LIN {X 0.182,Y -586.675,Z 1367.217,A 0.000,B 0.000,C 90.000,E1 75.102} C_DIS
LIN {X -0.131,Y -587.577,Z 1367.210,A 0.000,B 0.000,C 90.000,E1 73.795} C_DIS
LIN {X -0.025,Y -588.600,Z 1367.201,A 0.000,B 0.000,C 90.000,E1 72.181} C_DIS
LIN {X 0.175,Y -589.174,Z 1367.195,A 0.000,B 0.000,C 90.000,E1 71.094} C_DIS
LIN {X -0.190,Y -590.267,Z 1367.185,A 0.000,B 0.000,C 90.000,E1 69.263} C_DIS
LIN {X 0.230,Y -591.450,Z 1367.174,A 0.000,B 0.000,C 90.000,E1 67.358} C_DIS
LIN {X -0.084,Y -592.660,Z 1367.166,A 0.000,B 0.000,C 90.000,E1 65.793} C_DIS
LIN {X -0.029,Y -593.812,Z 1367.158,A 0.000,B 0.000,C 90.000,E1 64.460} C_DIS
LIN {X -0.046,Y -594.956,Z 1367.149,A 0.000,B 0.000,C 90.000,E1 62.871} C_DIS
LIN {X 0.337,Y -596.678,Z 1367.138,A 0.000,B 0.000,C 90.000,E1 60.717} C_DIS
LIN {X 0.286,Y -597.682,Z 1367.132,A 0.000,B 0.000,C 90.000,E1 59.665} C_DIS
LIN {X -0.217,Y -599.480,Z 1367.121,A 0.000,B 0.000,C 90.000,E1 57.867} C_DIS
LIN {X 0.070,Y -600.420,Z 1367.116,A 0.000,B 0.000,C 90.000,E1 56.786} C_DIS
LIN {X 0.111,Y -601.675,Z 1367.108,A 0.000,B 0.000,C 90.000,E1 55.468} C_DIS
LIN {X -0.317,Y -602.919,Z 1367.101,A 0.000,B 0.000,C 90.000,E1 54.196} C_DIS
LIN {X -0.207,Y -604.569,Z 1367.091,A 0.000,B 0.000,C 90.000,E1 52.351} C_DIS
LIN {X -0.112,Y -605.339,Z 1367.085,A 0.000,B 0.000,C 90.000,E1 51.295} C_DIS
LIN {X -0.057,Y -606.339,Z 1367.075,A 0.000,B 0.000,C 90.000,E1 49.461} C_DIS
LIN {X 0.070,Y -606.805,Z 1367.069,A 0.000,B 0.000,C 90.000,E1 48.405} C_DIS
LIN {X 0.003,Y -607.133,Z 1367.062,A 0.000,B 0.000,C 90.000,E1 47.106} C_DIS
LIN {X -0.086,Y -607.336,Z 1367.055,A 0.000,B 0.000,C 90.000,E1 45.810} C_DIS
LIN {X -0.164,Y -607.214,Z 1367.047,A 0.000,B 0.000,C 90.000,E1 44.514} C_DIS
LIN {X -0.060,Y -606.926,Z 1367.042,A 0.000,B 0.000,C 90.000,E1 43.461} C_DIS
LIN {X -0.317,Y -606.188,Z 1367.033,A 0.000,B 0.000,C 90.000,E1 41.919} C_DIS
LIN {X -0.191,Y -605.656,Z 1367.027,A 0.000,B 0.000,C 90.000,E1 40.862} C_DIS
LIN {X -0.274,Y -604.805,Z 1367.020,A 0.000,B 0.000,C 90.000,E1 39.564} C_DIS
LIN {X 0.036,Y -604.233,Z 1367.015,A 0.000,B 0.000,C 90.000,E1 38.749} C_DIS
LIN {X 0.006,Y -603.104,Z 1367.008,A 0.000,B 0.000,C 90.000,E1 37.443} C_DIS
LIN {X 0.185,Y -601.962,Z 1367.002,A 0.000,B 0.000,C 90.000,E1 36.377} C_DIS
LIN {X -0.151,Y -601.213,Z 1366.999,A 0.000,B 0.000,C 90.000,E1 35.884} C_DIS
LIN {X 0.000,Y -599.501,Z 1366.994,A 0.000,B 0.000,C 90.000,E1 34.818} C_DIS
LIN {X 0.014,Y -596.707,Z 1366.986,A 0.000,B 0.000,C 90.000,E1 33.499} C_DIS
LIN {X 0.259,Y -594.134,Z 1366.980,A 0.000,B 0.000,C 90.000,E1 32.418} C_DIS
LIN {X -0.241,Y -591.891,Z 1366.976,A 0.000,B 0.000,C 90.000,E1 31.671} C_DIS
LIN {X -0.146,Y -590.279,Z 1366.973,A 0.000,B 0.000,C 90.000,E1 31.131} C_DIS
LIN {X 0.001,Y -586.439,Z 1366.967,A 0.000,B 0.000,C 90.000,E1 30.050} C_DIS
LIN {X -0.076,Y -583.279,Z 1366.963,A 0.000,B 0.000,C 90.000,E1 29.255} C_DIS
LIN {X 0.110,Y -580.242,Z 1366.959,A 0.000,B 0.000,C 90.000,E1 28.565} C_DIS
LIN {X 0.037,Y -576.987,Z 1366.955,A 0.000,B 0.000,C 90.000,E1 27.897} C_DIS
LIN {X 0.097,Y -572.727,Z 1366.951,A 0.000,B 0.000,C 90.000,E1 27.078} C_DIS
LIN {X -0.054,Y -568.945,Z 1366.947,A 0.000,B 0.000,C 90.000,E1 26.411} C_DIS
LIN {X 0.018,Y -564.798,Z 1366.943,A 0.000,B 0.000,C 90.000,E1 25.720} C_DIS
LIN {X 0.152,Y -561.285,Z 1366.940,A 0.000,B 0.000,C 90.000,E1 25.155} C_DIS
LIN {X 0.054,Y -555.570,Z 1366.935,A 0.000,B 0.000,C 90.000,E1 24.335} C_DIS
LIN {X 0.134,Y -550.552,Z 1366.932,A 0.000,B 0.000,C 90.000,E1 23.643} C_DIS
LIN {X 0.165,Y -546.171,Z 1366.928,A 0.000,B 0.000,C 90.000,E1 23.078} C_DIS
LIN {X 0.114,Y -540.423,Z 1366.924,A 0.000,B 0.000,C 90.000,E1 22.386} C_DIS
LIN {X -0.268,Y -534.283,Z 1366.921,A 0.000,B 0.000,C 90.000,E1 21.716} C_DIS
LIN {X 0.001,Y -523.934,Z 1366.914,A 0.000,B 0.000,C 90.000,E1 20.556} C_DIS
LIN {X -0.191,Y -511.865,Z 1366.907,A 0.000,B 0.000,C 90.000,E1 19.322} C_DIS
LIN {X -0.080,Y -502.797,Z 1366.902,A 0.000,B 0.000,C 90.000,E1 18.362} C_DIS
LIN {X -0.238,Y -493.197,Z 1366.897,A 0.000,B 0.000,C 90.000,E1 17.402} C_DIS
LIN {X 0.136,Y -480.687,Z 1366.890,A 0.000,B 0.000,C 90.000,E1 16.134} C_DIS
LIN {X 0.231,Y -465.377,Z 1366.881,A 0.000,B 0.000,C 90.000,E1 14.592} C_DIS
LIN {X -0.148,Y -455.458,Z 1366.876,A 0.000,B 0.000,C 90.000,E1 13.647} C_DIS
LIN {X -0.104,Y -438.414,Z 1366.866,A 0.000,B 0.000,C 90.000,E1 11.883} C_DIS
LIN {X 0.074,Y -430.022,Z 1366.861,A 0.000,B 0.000,C 90.000,E1 10.950} C_DIS
LIN {X 0.023,Y -416.118,Z 1366.852,A 0.000,B 0.000,C 90.000,E1 9.378} C_DIS
LIN {X -0.121,Y -403.557,Z 1366.844,A 0.000,B 0.000,C 90.000,E1 7.936} C_DIS
LIN {X 0.155,Y -397.824,Z 1366.840,A 0.000,B 0.000,C 90.000,E1 7.239} C_DIS
LIN {X -0.185,Y -392.988,Z 1366.837,A 0.000,B 0.000,C 90.000,E1 6.606} C_DIS
LIN {X 0.034,Y -392.603,Z 1366.836,A 0.000,B 0.000,C 90.000,E1 6.486} C_DIS
LIN {X -0.004,Y -392.597,Z 1366.836,A 0.000,B 0.000,C 90.000,E1 6.486} C_DIS
LIN {X 0.166,Y -394.316,Z 1366.835,A 0.000,B 0.000,C 90.000,E1 6.201} C_DIS
LIN {X -0.174,Y -398.130,Z 1366.833,A 0.000,B 0.000,C 90.000,E1 5.910} C_DIS
LIN {X -0.140,Y -408.338,Z 1366.829,A 0.000,B 0.000,C 90.000,E1 5.163} C_DIS
LIN {X -0.103,Y -415.972,Z 1366.825,A 0.000,B 0.000,C 90.000,E1 4.531} C_DIS
LIN {X -0.114,Y -420.296,Z 1366.823,A 0.000,B 0.000,C 90.000,E1 4.131} C_DIS
LIN {X 0.071,Y -424.536,Z 1366.820,A 0.000,B 0.000,C 90.000,E1 3.669} C_DIS
LIN {X 0.122,Y -430.041,Z 1366.817,A 0.000,B 0.000,C 90.000,E1 3.037} C_DIS
LIN {X -0.080,Y -435.402,Z 1366.813,A 0.000,B 0.000,C 90.000,E1 2.407} C_DIS
LIN {X 0.212,Y -441.815,Z 1366.809,A 0.000,B 0.000,C 90.000,E1 1.547} C_DIS
LIN {X 0.086,Y -447.840,Z 1366.804,A 0.000,B 0.000,C 90.000,E1 0.745} C_DIS
LIN {X 0.000,Y -453.201,Z 1366.800,A 0.000,B 0.000,C 90.000,E1 360.000} C_DIS
LIN {X 0.073,Y -458.775,Z 1366.795,A 0.000,B 0.000,C 90.000,E1 359.141} C_DIS
LIN {X 0.003,Y -462.817,Z 1366.792,A 0.000,B 0.000,C 90.000,E1 358.511} C_DIS
LIN {X 0.204,Y -468.275,Z 1366.786,A 0.000,B 0.000,C 90.000,E1 357.535} C_DIS
LIN {X 0.203,Y -471.754,Z 1366.783,A 0.000,B 0.000,C 90.000,E1 356.906} C_DIS
LIN {X -0.091,Y -475.709,Z 1366.779,A 0.000,B 0.000,C 90.000,E1 356.159} C_DIS
LIN {X 0.125,Y -479.359,Z 1366.774,A 0.000,B 0.000,C 90.000,E1 355.355} C_DIS
LIN {X -0.101,Y -482.673,Z 1366.770,A 0.000,B 0.000,C 90.000,E1 354.609} C_DIS
LIN {X -0.109,Y -484.570,Z 1366.767,A 0.000,B 0.000,C 90.000,E1 354.147} C_DIS
LIN {X -0.093,Y -487.981,Z 1366.762,A 0.000,B 0.000,C 90.000,E1 353.223} C_DIS
LIN {X -0.039,Y -491.080,Z 1366.757,A 0.000,B 0.000,C 90.000,E1 352.299} C_DIS
LIN {X 0.226,Y -492.982,Z 1366.754,A 0.000,B 0.000,C 90.000,E1 351.659} C_DIS
LIN {X -0.054,Y -494.713,Z 1366.750,A 0.000,B 0.000,C 90.000,E1 351.084} C_DIS
LIN {X 0.154,Y -497.020,Z 1366.745,A 0.000,B 0.000,C 90.000,E1 350.151} C_DIS
LIN {X -0.096,Y -499.120,Z 1366.740,A 0.000,B 0.000,C 90.000,E1 349.275} C_DIS
LIN {X 0.096,Y -501.580,Z 1366.734,A 0.000,B 0.000,C 90.000,E1 348.049} C_DIS
LIN {X -0.042,Y -502.671,Z 1366.730,A 0.000,B 0.000,C 90.000,E1 347.465} C_DIS
LIN {X -0.183,Y -504.702,Z 1366.724,A 0.000,B 0.000,C 90.000,E1 346.284} C_DIS
LIN {X 0.187,Y -505.538,Z 1366.720,A 0.000,B 0.000,C 90.000,E1 345.644} C_DIS
LIN {X 0.127,Y -505.707,Z 1366.719,A 0.000,B 0.000,C 90.000,E1 345.353} C_DIS
LIN {X 0.198,Y -505.709,Z 1366.717,A 0.000,B 0.000,C 90.000,E1 345.046} C_DIS
LIN {X 0.139,Y -505.490,Z 1366.715,A 0.000,B 0.000,C 90.000,E1 344.755} C_DIS
LIN {X 0.078,Y -504.841,Z 1366.714,A 0.000,B 0.000,C 90.000,E1 344.464} C_DIS
LIN {X -0.128,Y -504.230,Z 1366.713,A 0.000,B 0.000,C 90.000,E1 344.338} C_DIS
LIN {X 0.152,Y -503.084,Z 1366.712,A 0.000,B 0.000,C 90.000,E1 344.157} C_DIS
LIN {X 0.156,Y -499.851,Z 1366.711,A 0.000,B 0.000,C 90.000,E1 344.031} C_DIS
LIN {X -0.040,Y -466.644,Z 1366.705,A 0.000,B 0.000,C 90.000,E1 342.906} C_DIS
LIN {X 0.169,Y -435.494,Z 1366.698,A 0.000,B 0.000,C 90.000,E1 341.638} C_DIS
LIN {X -0.147,Y -408.031,Z 1366.691,A 0.000,B 0.000,C 90.000,E1 340.423} C_DIS
LIN {X -0.120,Y -382.486,Z 1366.684,A 0.000,B 0.000,C 90.000,E1 339.082} C_DIS
LIN {X 0.064,Y -362.176,Z 1366.677,A 0.000,B 0.000,C 90.000,E1 337.847} C_DIS
LIN {X 0.043,Y -362.174,Z 1366.677,A 0.000,B 0.000,C 90.000,E1 337.847} C_DIS
LIN {X 0.164,Y -366.198,Z 1366.641,A 0.000,B 0.000,C 90.000,E1 331.385} C_DIS
LIN {X -0.133,Y -371.227,Z 1366.604,A 0.000,B 0.000,C 90.000,E1 324.769} C_DIS
LIN {X -0.146,Y -371.660,Z 1366.602,A 0.000,B 0.000,C 90.000,E1 324.402} C_DIS
LIN {X -0.090,Y -376.765,Z 1366.570,A 0.000,B 0.000,C 90.000,E1 318.528} C_DIS
LIN {X 0.200,Y -378.156,Z 1366.563,A 0.000,B 0.000,C 90.000,E1 317.391} C_DIS
LIN {X -0.061,Y -384.283,Z 1366.529,A 0.000,B 0.000,C 90.000,E1 311.272} C_DIS
LIN {X -0.019,Y -384.786,Z 1366.527,A 0.000,B 0.000,C 90.000,E1 310.906} C_DIS
LIN {X -0.029,Y -390.954,Z 1366.493,A 0.000,B 0.000,C 90.000,E1 304.818} C_DIS
LIN {X 0.038,Y -391.366,Z 1366.491,A 0.000,B 0.000,C 90.000,E1 304.452} C_DIS
LIN {X -0.232,Y -396.686,Z 1366.460,A 0.000,B 0.000,C 90.000,E1 298.821} C_DIS
LIN {X -0.014,Y -397.074,Z 1366.458,A 0.000,B 0.000,C 90.000,E1 298.437} C_DIS
LIN {X -0.058,Y -401.487,Z 1366.427,A 0.000,B 0.000,C 90.000,E1 292.823} C_DIS
LIN {X 0.108,Y -401.768,Z 1366.423,A 0.000,B 0.000,C 90.000,E1 292.099} C_DIS
LIN {X 0.068,Y -404.565,Z 1366.396,A 0.000,B 0.000,C 90.000,E1 287.221} C_DIS
LIN {X 0.170,Y -404.760,Z 1366.394,A 0.000,B 0.000,C 90.000,E1 286.858} C_DIS
LIN {X 0.077,Y -406.039,Z 1366.365,A 0.000,B 0.000,C 90.000,E1 281.658} C_DIS
LIN {X 0.166,Y -406.138,Z 1366.363,A 0.000,B 0.000,C 90.000,E1 281.299} C_DIS
LIN {X -0.207,Y -405.655,Z 1366.334,A 0.000,B 0.000,C 90.000,E1 276.144} C_DIS
LIN {X 0.201,Y -405.601,Z 1366.332,A 0.000,B 0.000,C 90.000,E1 275.739} C_DIS
LIN {X -0.129,Y -403.549,Z 1366.305,A 0.000,B 0.000,C 90.000,E1 270.917} C_DIS
LIN {X -0.194,Y -403.040,Z 1366.301,A 0.000,B 0.000,C 90.000,E1 270.229} C_DIS
LIN {X 0.031,Y -399.011,Z 1366.272,A 0.000,B 0.000,C 90.000,E1 264.951} C_DIS
LIN {X -0.143,Y -397.175,Z 1366.264,A 0.000,B 0.000,C 90.000,E1 263.571} C_DIS
LIN {X -0.194,Y -392.923,Z 1366.241,A 0.000,B 0.000,C 90.000,E1 259.342} C_DIS
LIN {X 0.182,Y -391.869,Z 1366.237,A 0.000,B 0.000,C 90.000,E1 258.578} C_DIS
LIN {X -0.062,Y -385.732,Z 1366.211,A 0.000,B 0.000,C 90.000,E1 253.976} C_DIS
LIN {X -0.127,Y -384.968,Z 1366.207,A 0.000,B 0.000,C 90.000,E1 253.268} C_DIS
LIN {X 0.100,Y -378.113,Z 1366.183,A 0.000,B 0.000,C 90.000,E1 248.901} C_DIS
LIN {X -0.164,Y -376.355,Z 1366.175,A 0.000,B 0.000,C 90.000,E1 247.486} C_DIS
LIN {X -0.038,Y -375.852,Z 1366.173,A 0.000,B 0.000,C 90.000,E1 247.102} C_DIS
LIN {X -0.088,Y -369.083,Z 1366.150,A 0.000,B 0.000,C 90.000,E1 243.076} C_DIS
LIN {X -0.009,Y -366.236,Z 1366.138,A 0.000,B 0.000,C 90.000,E1 240.845} C_DIS
LIN {X -0.047,Y -358.830,Z 1366.113,A 0.000,B 0.000,C 90.000,E1 236.373} C_DIS
LIN {X -0.059,Y -356.022,Z 1366.101,A 0.000,B 0.000,C 90.000,E1 234.116} C_DIS
LIN {X -0.062,Y -348.459,Z 1366.073,A 0.000,B 0.000,C 90.000,E1 229.175} C_DIS
LIN {X -0.001,Y -345.873,Z 1366.060,A 0.000,B 0.000,C 90.000,E1 226.863} C_DIS
LIN {X -0.033,Y -339.106,Z 1366.032,A 0.000,B 0.000,C 90.000,E1 221.838} C_DIS
LIN {X 0.051,Y -336.944,Z 1366.019,A 0.000,B 0.000,C 90.000,E1 219.483} C_DIS
LIN {X 0.031,Y -331.620,Z 1365.993,A 0.000,B 0.000,C 90.000,E1 214.771} C_DIS
LIN {X 0.101,Y -329.361,Z 1365.976,A 0.000,B 0.000,C 90.000,E1 211.592} C_DIS
LIN {X 0.113,Y -328.630,Z 1365.971,A 0.000,B 0.000,C 90.000,E1 210.797} C_DIS
LIN {X -0.181,Y -324.550,Z 1365.940,A 0.000,B 0.000,C 90.000,E1 205.283} C_DIS
LIN {X -0.199,Y -324.574,Z 1365.940,A 0.000,B 0.000,C 90.000,E1 205.283} C_DIS
LIN {X -0.065,Y -343.510,Z 1365.932,A 0.000,B 0.000,C 90.000,E1 203.823} C_DIS
LIN {X 0.111,Y -364.170,Z 1365.925,A 0.000,B 0.000,C 90.000,E1 202.408} C_DIS
LIN {X -0.078,Y -386.764,Z 1365.917,A 0.000,B 0.000,C 90.000,E1 201.099} C_DIS
LIN {X 0.144,Y -413.035,Z 1365.910,A 0.000,B 0.000,C 90.000,E1 199.704} C_DIS
LIN {X 0.218,Y -441.275,Z 1365.902,A 0.000,B 0.000,C 90.000,E1 198.417} C_DIS
LIN {X -0.100,Y -446.323,Z 1365.901,A 0.000,B 0.000,C 90.000,E1 198.236} C_DIS
LIN {X 0.088,Y -447.679,Z 1365.900,A 0.000,B 0.000,C 90.000,E1 198.055} C_DIS
LIN {X 0.266,Y -448.506,Z 1365.900,A 0.000,B 0.000,C 90.000,E1 197.873} C_DIS
LIN {X -0.122,Y -449.127,Z 1365.899,A 0.000,B 0.000,C 90.000,E1 197.764} C_DIS
LIN {X 0.177,Y -450.069,Z 1365.897,A 0.000,B 0.000,C 90.000,E1 197.402} C_DIS
LIN {X 0.048,Y -450.694,Z 1365.895,A 0.000,B 0.000,C 90.000,E1 197.094} C_DIS
LIN {X -0.210,Y -451.133,Z 1365.893,A 0.000,B 0.000,C 90.000,E1 196.804} C_DIS
LIN {X 0.155,Y -451.880,Z 1365.888,A 0.000,B 0.000,C 90.000,E1 195.788} C_DIS
LIN {X 0.045,Y -453.011,Z 1365.879,A 0.000,B 0.000,C 90.000,E1 194.189} C_DIS
LIN {X 0.188,Y -453.802,Z 1365.872,A 0.000,B 0.000,C 90.000,E1 192.883} C_DIS
LIN {X -0.002,Y -454.650,Z 1365.863,A 0.000,B 0.000,C 90.000,E1 191.299} C_DIS
LIN {X -0.036,Y -455.227,Z 1365.856,A 0.000,B 0.000,C 90.000,E1 190.018} C_DIS
LIN {X -0.134,Y -455.673,Z 1365.849,A 0.000,B 0.000,C 90.000,E1 188.746} C_DIS
LIN {X 0.075,Y -455.919,Z 1365.843,A 0.000,B 0.000,C 90.000,E1 187.757} C_DIS
LIN {X -0.081,Y -456.266,Z 1365.833,A 0.000,B 0.000,C 90.000,E1 185.853} C_DIS
LIN {X 0.028,Y -456.324,Z 1365.827,A 0.000,B 0.000,C 90.000,E1 184.878} C_DIS
LIN {X -0.101,Y -456.190,Z 1365.820,A 0.000,B 0.000,C 90.000,E1 183.612} C_DIS
LIN {X 0.011,Y -455.960,Z 1365.815,A 0.000,B 0.000,C 90.000,E1 182.636} C_DIS
LIN {X -0.080,Y -455.745,Z 1365.811,A 0.000,B 0.000,C 90.000,E1 182.007} C_DIS
LIN {X 0.023,Y -455.119,Z 1365.806,A 0.000,B 0.000,C 90.000,E1 181.031} C_DIS
LIN {X -0.072,Y -454.546,Z 1365.802,A 0.000,B 0.000,C 90.000,E1 180.401} C_DIS
LIN {X -0.169,Y -453.770,Z 1365.799,A 0.000,B 0.000,C 90.000,E1 179.771} C_DIS
LIN {X 0.067,Y -451.689,Z 1365.792,A 0.000,B 0.000,C 90.000,E1 178.453} C_DIS
LIN {X -0.039,Y -450.487,Z 1365.788,A 0.000,B 0.000,C 90.000,E1 177.822} C_DIS
LIN {X 0.123,Y -449.773,Z 1365.786,A 0.000,B 0.000,C 90.000,E1 177.478} C_DIS
LIN {X -0.169,Y -448.926,Z 1365.784,A 0.000,B 0.000,C 90.000,E1 177.192} C_DIS
LIN {X -0.144,Y -445.871,Z 1365.779,A 0.000,B 0.000,C 90.000,E1 176.216} C_DIS
LIN {X 0.158,Y -443.707,Z 1365.775,A 0.000,B 0.000,C 90.000,E1 175.527} C_DIS
LIN {X 0.000,Y -440.751,Z 1365.772,A 0.000,B 0.000,C 90.000,E1 174.894} C_DIS
LIN {X 0.204,Y -438.571,Z 1365.769,A 0.000,B 0.000,C 90.000,E1 174.375} C_DIS
LIN {X 0.049,Y -434.159,Z 1365.764,A 0.000,B 0.000,C 90.000,E1 173.571} C_DIS
LIN {X -0.218,Y -431.237,Z 1365.762,A 0.000,B 0.000,C 90.000,E1 173.109} C_DIS
LIN {X 0.032,Y -425.872,Z 1365.757,A 0.000,B 0.000,C 90.000,E1 172.243} C_DIS
LIN {X -0.194,Y -420.132,Z 1365.752,A 0.000,B 0.000,C 90.000,E1 171.432} C_DIS
LIN {X 0.101,Y -406.286,Z 1365.741,A 0.000,B 0.000,C 90.000,E1 169.342} C_DIS
LIN {X 0.216,Y -393.490,Z 1365.729,A 0.000,B 0.000,C 90.000,E1 167.229} C_DIS
LIN {X 0.198,Y -390.708,Z 1365.726,A 0.000,B 0.000,C 90.000,E1 166.700} C_DIS
LIN {X -0.069,Y -387.799,Z 1365.722,A 0.000,B 0.000,C 90.000,E1 165.936} C_DIS
LIN {X -0.087,Y -387.536,Z 1365.719,A 0.000,B 0.000,C 90.000,E1 165.408} C_DIS
LIN {X -0.125,Y -387.556,Z 1365.719,A 0.000,B 0.000,C 90.000,E1 165.408} C_DIS
LIN {X -0.135,Y -388.274,Z 1365.718,A 0.000,B 0.000,C 90.000,E1 165.227} C_DIS
LIN {X -0.128,Y -392.971,Z 1365.714,A 0.000,B 0.000,C 90.000,E1 164.574} C_DIS
LIN {X -0.108,Y -399.230,Z 1365.710,A 0.000,B 0.000,C 90.000,E1 163.866} C_DIS
LIN {X -0.180,Y -408.697,Z 1365.705,A 0.000,B 0.000,C 90.000,E1 162.960} C_DIS
LIN {X 0.013,Y -425.885,Z 1365.697,A 0.000,B 0.000,C 90.000,E1 161.456} C_DIS
LIN {X 0.257,Y -449.800,Z 1365.687,A 0.000,B 0.000,C 90.000,E1 159.571} C_DIS
LIN {X -0.100,Y -459.141,Z 1365.683,A 0.000,B 0.000,C 90.000,E1 158.901} C_DIS
LIN {X -0.021,Y -466.703,Z 1365.679,A 0.000,B 0.000,C 90.000,E1 158.284} C_DIS
LIN {X -0.108,Y -472.655,Z 1365.677,A 0.000,B 0.000,C 90.000,E1 157.794} C_DIS
LIN {X -0.283,Y -481.389,Z 1365.672,A 0.000,B 0.000,C 90.000,E1 157.050} C_DIS
LIN {X -0.124,Y -489.927,Z 1365.668,A 0.000,B 0.000,C 90.000,E1 156.230} C_DIS
LIN {X 0.098,Y -495.512,Z 1365.665,A 0.000,B 0.000,C 90.000,E1 155.665} C_DIS
LIN {X 0.218,Y -500.943,Z 1365.662,A 0.000,B 0.000,C 90.000,E1 155.101} C_DIS
LIN {X -0.117,Y -504.951,Z 1365.660,A 0.000,B 0.000,C 90.000,E1 154.717} C_DIS
LIN {X -0.091,Y -512.632,Z 1365.655,A 0.000,B 0.000,C 90.000,E1 153.845} C_DIS
LIN {X -0.256,Y -518.709,Z 1365.651,A 0.000,B 0.000,C 90.000,E1 153.127} C_DIS
LIN {X 0.082,Y -524.193,Z 1365.646,A 0.000,B 0.000,C 90.000,E1 152.359} C_DIS
LIN {X -0.238,Y -526.299,Z 1365.645,A 0.000,B 0.000,C 90.000,E1 152.103} C_DIS
LIN {X -0.145,Y -530.043,Z 1365.642,A 0.000,B 0.000,C 90.000,E1 151.513} C_DIS
LIN {X -0.170,Y -533.906,Z 1365.638,A 0.000,B 0.000,C 90.000,E1 150.795} C_DIS
LIN {X -0.019,Y -536.557,Z 1365.635,A 0.000,B 0.000,C 90.000,E1 150.205} C_DIS
LIN {X 0.144,Y -539.972,Z 1365.630,A 0.000,B 0.000,C 90.000,E1 149.331} C_DIS
LIN {X -0.127,Y -541.955,Z 1365.627,A 0.000,B 0.000,C 90.000,E1 148.791} C_DIS
LIN {X 0.079,Y -543.704,Z 1365.623,A 0.000,B 0.000,C 90.000,E1 148.201} C_DIS
LIN {X -0.140,Y -545.900,Z 1365.619,A 0.000,B 0.000,C 90.000,E1 147.375} C_DIS
LIN {X 0.089,Y -547.150,Z 1365.616,A 0.000,B 0.000,C 90.000,E1 146.786} C_DIS
LIN {X -0.049,Y -549.147,Z 1365.609,A 0.000,B 0.000,C 90.000,E1 145.674} C_DIS
LIN {X 0.106,Y -550.435,Z 1365.605,A 0.000,B 0.000,C 90.000,E1 144.815} C_DIS
LIN {X 0.017,Y -551.761,Z 1365.598,A 0.000,B 0.000,C 90.000,E1 143.703} C_DIS
LIN {X 0.269,Y -552.794,Z 1365.592,A 0.000,B 0.000,C 90.000,E1 142.557} C_DIS
LIN {X 0.099,Y -553.616,Z 1365.586,A 0.000,B 0.000,C 90.000,E1 141.457} C_DIS
LIN {X 0.076,Y -554.674,Z 1365.577,A 0.000,B 0.000,C 90.000,E1 139.784} C_DIS
LIN {X -0.068,Y -555.526,Z 1365.569,A 0.000,B 0.000,C 90.000,E1 138.405} C_DIS
LIN {X -0.162,Y -556.345,Z 1365.560,A 0.000,B 0.000,C 90.000,E1 136.743} C_DIS
LIN {X 0.107,Y -556.913,Z 1365.552,A 0.000,B 0.000,C 90.000,E1 135.324} C_DIS
LIN {X 0.093,Y -557.710,Z 1365.541,A 0.000,B 0.000,C 90.000,E1 133.380} C_DIS
LIN {X 0.113,Y -558.710,Z 1365.530,A 0.000,B 0.000,C 90.000,E1 131.434} C_DIS
LIN {X -0.271,Y -559.658,Z 1365.526,A 0.000,B 0.000,C 90.000,E1 130.620} C_DIS
LIN {X -0.312,Y -559.675,Z 1365.526,A 0.000,B 0.000,C 90.000,E1 130.620} C_DIS
LIN {X 0.204,Y -560.719,Z 1365.525,A 0.000,B 0.000,C 90.000,E1 130.458} C_DIS
LIN {X 0.111,Y -561.623,Z 1365.524,A 0.000,B 0.000,C 90.000,E1 130.334} C_DIS
LIN {X 0.127,Y -562.227,Z 1365.523,A 0.000,B 0.000,C 90.000,E1 130.172} C_DIS
LIN {X 0.084,Y -562.282,Z 1365.523,A 0.000,B 0.000,C 90.000,E1 130.172} C_DIS
LIN {X -0.227,Y -564.588,Z 1365.523,A 0.000,B 0.000,C 90.000,E1 130.092} C_DIS
LIN {X -0.283,Y -566.188,Z 1365.522,A 0.000,B 0.000,C 90.000,E1 130.011} C_DIS
LIN {X 0.133,Y -574.296,Z 1365.521,A 0.000,B 0.000,C 90.000,E1 129.725} C_DIS
LIN {X 0.261,Y -579.457,Z 1365.520,A 0.000,B 0.000,C 90.000,E1 129.564} C_DIS
LIN {X 0.015,Y -581.996,Z 1365.519,A 0.000,B 0.000,C 90.000,E1 129.483} C_DIS
LIN {X -0.148,Y -585.029,Z 1365.519,A 0.000,B 0.000,C 90.000,E1 129.358} C_DIS
LIN {X 0.191,Y -590.891,Z 1365.517,A 0.000,B 0.000,C 90.000,E1 128.991} C_DIS
LIN {X -0.248,Y -595.306,Z 1365.515,A 0.000,B 0.000,C 90.000,E1 128.749} C_DIS
LIN {X 0.028,Y -600.950,Z 1365.513,A 0.000,B 0.000,C 90.000,E1 128.302} C_DIS
LIN {X 0.020,Y -606.411,Z 1365.510,A 0.000,B 0.000,C 90.000,E1 127.855} C_DIS
LIN {X -0.070,Y -612.969,Z 1365.507,A 0.000,B 0.000,C 90.000,E1 127.282} C_DIS
LIN {X -0.062,Y -616.756,Z 1365.505,A 0.000,B 0.000,C 90.000,E1 126.916} C_DIS
LIN {X 0.200,Y -625.260,Z 1365.500,A 0.000,B 0.000,C 90.000,E1 126.011} C_DIS
LIN {X -0.098,Y -628.604,Z 1365.498,A 0.000,B 0.000,C 90.000,E1 125.678} C_DIS
LIN {X 0.102,Y -635.118,Z 1365.494,A 0.000,B 0.000,C 90.000,E1 124.898} C_DIS
LIN {X -0.011,Y -640.076,Z 1365.490,A 0.000,B 0.000,C 90.000,E1 124.278} C_DIS
LIN {X 0.098,Y -643.801,Z 1365.488,A 0.000,B 0.000,C 90.000,E1 123.785} C_DIS
LIN {X 0.058,Y -648.265,Z 1365.484,A 0.000,B 0.000,C 90.000,E1 123.166} C_DIS
LIN {X 0.051,Y -652.359,Z 1365.481,A 0.000,B 0.000,C 90.000,E1 122.546} C_DIS
LIN {X -0.369,Y -654.670,Z 1365.479,A 0.000,B 0.000,C 90.000,E1 122.212} C_DIS
LIN {X -0.133,Y -658.591,Z 1365.475,A 0.000,B 0.000,C 90.000,E1 121.465} C_DIS
LIN {X 0.040,Y -660.427,Z 1365.473,A 0.000,B 0.000,C 90.000,E1 121.082} C_DIS
LIN {X 0.188,Y -663.616,Z 1365.469,A 0.000,B 0.000,C 90.000,E1 120.335} C_DIS
LIN {X 0.029,Y -666.155,Z 1365.465,A 0.000,B 0.000,C 90.000,E1 119.617} C_DIS
LIN {X 0.221,Y -668.142,Z 1365.461,A 0.000,B 0.000,C 90.000,E1 118.871} C_DIS
LIN {X 0.375,Y -668.696,Z 1365.459,A 0.000,B 0.000,C 90.000,E1 118.615} C_DIS
LIN {X 0.263,Y -669.704,Z 1365.455,A 0.000,B 0.000,C 90.000,E1 117.897} C_DIS
LIN {X -0.147,Y -669.966,Z 1365.451,A 0.000,B 0.000,C 90.000,E1 117.206} C_DIS
LIN {X -0.247,Y -669.843,Z 1365.447,A 0.000,B 0.000,C 90.000,E1 116.488} C_DIS
LIN {X 0.248,Y -669.374,Z 1365.443,A 0.000,B 0.000,C 90.000,E1 115.720} C_DIS
LIN {X -0.154,Y -668.585,Z 1365.439,A 0.000,B 0.000,C 90.000,E1 115.027} C_DIS
LIN {X 0.006,Y -668.253,Z 1365.438,A 0.000,B 0.000,C 90.000,E1 114.771} C_DIS
LIN {X 0.047,Y -666.989,Z 1365.435,A 0.000,B 0.000,C 90.000,E1 114.283} C_DIS
LIN {X 0.203,Y -666.014,Z 1365.434,A 0.000,B 0.000,C 90.000,E1 114.027} C_DIS
LIN {X -0.109,Y -663.067,Z 1365.431,A 0.000,B 0.000,C 90.000,E1 113.567} C_DIS
LIN {X -0.040,Y -662.029,Z 1365.430,A 0.000,B 0.000,C 90.000,E1 113.439} C_DIS
LIN {X -0.147,Y -656.469,Z 1365.428,A 0.000,B 0.000,C 90.000,E1 113.003} C_DIS
LIN {X -0.180,Y -654.733,Z 1365.427,A 0.000,B 0.000,C 90.000,E1 112.898} C_DIS
LIN {X -0.185,Y -648.596,Z 1365.426,A 0.000,B 0.000,C 90.000,E1 112.642} C_DIS
LIN {X -0.187,Y -644.606,Z 1365.425,A 0.000,B 0.000,C 90.000,E1 112.514} C_DIS
LIN {X -0.066,Y -634.954,Z 1365.424,A 0.000,B 0.000,C 90.000,E1 112.259} C_DIS
LIN {X 0.181,Y -629.604,Z 1365.423,A 0.000,B 0.000,C 90.000,E1 112.099} C_DIS
LIN {X 0.126,Y -629.435,Z 1365.423,A 0.000,B 0.000,C 90.000,E1 112.099} C_DIS
LIN {X -0.146,Y -630.466,Z 1365.422,A 0.000,B 0.000,C 90.000,E1 111.972} C_DIS
LIN {X -0.274,Y -639.281,Z 1365.416,A 0.000,B 0.000,C 90.000,E1 110.972} C_DIS
LIN {X -0.179,Y -643.249,Z 1365.414,A 0.000,B 0.000,C 90.000,E1 110.482} C_DIS
LIN {X 0.343,Y -647.430,Z 1365.410,A 0.000,B 0.000,C 90.000,E1 109.812} C_DIS
LIN {X 0.224,Y -649.628,Z 1365.408,A 0.000,B 0.000,C 90.000,E1 109.450} C_DIS
LIN {X -0.022,Y -653.008,Z 1365.405,A 0.000,B 0.000,C 90.000,E1 108.852} C_DIS
LIN {X -0.117,Y -657.558,Z 1365.399,A 0.000,B 0.000,C 90.000,E1 107.873} C_DIS
LIN {X 0.372,Y -660.755,Z 1365.395,A 0.000,B 0.000,C 90.000,E1 107.094} C_DIS
LIN {X 0.072,Y -663.615,Z 1365.391,A 0.000,B 0.000,C 90.000,E1 106.386} C_DIS
LIN {X -0.013,Y -666.033,Z 1365.387,A 0.000,B 0.000,C 90.000,E1 105.662} C_DIS
LIN {X -0.258,Y -667.873,Z 1365.383,A 0.000,B 0.000,C 90.000,E1 104.954} C_DIS
LIN {X 0.238,Y -668.850,Z 1365.380,A 0.000,B 0.000,C 90.000,E1 104.426} C_DIS
LIN {X 0.027,Y -669.855,Z 1365.376,A 0.000,B 0.000,C 90.000,E1 103.716} C_DIS
LIN {X -0.110,Y -670.297,Z 1365.374,A 0.000,B 0.000,C 90.000,E1 103.244} C_DIS
LIN {X -0.311,Y -670.497,Z 1365.370,A 0.000,B 0.000,C 90.000,E1 102.535} C_DIS
LIN {X 0.141,Y -670.333,Z 1365.365,A 0.000,B 0.000,C 90.000,E1 101.771} C_DIS
LIN {X 0.072,Y -670.208,Z 1365.364,A 0.000,B 0.000,C 90.000,E1 101.535} C_DIS
LIN {X -0.272,Y -669.384,Z 1365.360,A 0.000,B 0.000,C 90.000,E1 100.838} C_DIS
LIN {X 0.237,Y -668.657,Z 1365.357,A 0.000,B 0.000,C 90.000,E1 100.310} C_DIS
LIN {X -0.036,Y -667.668,Z 1365.355,A 0.000,B 0.000,C 90.000,E1 99.849} C_DIS
LIN {X -0.201,Y -666.410,Z 1365.352,A 0.000,B 0.000,C 90.000,E1 99.378} C_DIS
LIN {X 0.172,Y -664.934,Z 1365.349,A 0.000,B 0.000,C 90.000,E1 98.859} C_DIS
LIN {X -0.217,Y -662.224,Z 1365.345,A 0.000,B 0.000,C 90.000,E1 98.163} C_DIS
LIN {X 0.135,Y -660.250,Z 1365.343,A 0.000,B 0.000,C 90.000,E1 97.644} C_DIS
LIN {X -0.302,Y -656.924,Z 1365.339,A 0.000,B 0.000,C 90.000,E1 96.947} C_DIS
LIN {X 0.043,Y -655.113,Z 1365.336,A 0.000,B 0.000,C 90.000,E1 96.549} C_DIS
LIN {X -0.303,Y -652.457,Z 1365.334,A 0.000,B 0.000,C 90.000,E1 96.087} C_DIS
LIN {X -0.178,Y -647.963,Z 1365.330,A 0.000,B 0.000,C 90.000,E1 95.334} C_DIS
LIN {X -0.164,Y -643.191,Z 1365.325,A 0.000,B 0.000,C 90.000,E1 94.588} C_DIS
LIN {X -0.074,Y -638.959,Z 1365.322,A 0.000,B 0.000,C 90.000,E1 93.955} C_DIS
LIN {X 0.065,Y -635.128,Z 1365.319,A 0.000,B 0.000,C 90.000,E1 93.440} C_DIS
LIN {X 0.082,Y -629.543,Z 1365.316,A 0.000,B 0.000,C 90.000,E1 92.808} C_DIS
LIN {X 0.146,Y -623.401,Z 1365.312,A 0.000,B 0.000,C 90.000,E1 92.178} C_DIS
LIN {X 0.218,Y -615.720,Z 1365.308,A 0.000,B 0.000,C 90.000,E1 91.432} C_DIS
LIN {X -0.008,Y -611.713,Z 1365.306,A 0.000,B 0.000,C 90.000,E1 91.088} C_DIS
LIN {X -0.109,Y -607.317,Z 1365.304,A 0.000,B 0.000,C 90.000,E1 90.745} C_DIS
LIN {X 0.085,Y -602.939,Z 1365.302,A 0.000,B 0.000,C 90.000,E1 90.401} C_DIS
LIN {X 0.229,Y -596.196,Z 1365.300,A 0.000,B 0.000,C 90.000,E1 90.000} C_DIS
LIN {X -0.222,Y -589.332,Z 1365.298,A 0.000,B 0.000,C 90.000,E1 89.714} C_DIS
LIN {X -0.119,Y -584.030,Z 1365.297,A 0.000,B 0.000,C 90.000,E1 89.484} C_DIS
LIN {X 0.001,Y -578.143,Z 1365.296,A 0.000,B 0.000,C 90.000,E1 89.198} C_DIS
LIN {X -0.114,Y -574.268,Z 1365.294,A 0.000,B 0.000,C 90.000,E1 88.912} C_DIS
LIN {X -0.151,Y -574.243,Z 1365.294,A 0.000,B 0.000,C 90.000,E1 88.912} C_DIS
LIN {X -0.170,Y -573.640,Z 1365.293,A 0.000,B 0.000,C 90.000,E1 88.740} C_DIS
LIN {X -0.152,Y -573.457,Z 1365.292,A 0.000,B 0.000,C 90.000,E1 88.568} C_DIS
LIN {X -0.271,Y -573.745,Z 1365.288,A 0.000,B 0.000,C 90.000,E1 87.822} C_DIS
LIN {X -0.071,Y -575.894,Z 1365.274,A 0.000,B 0.000,C 90.000,E1 85.355} C_DIS
LIN {X -0.209,Y -577.628,Z 1365.265,A 0.000,B 0.000,C 90.000,E1 83.742} C_DIS
LIN {X -0.097,Y -579.909,Z 1365.255,A 0.000,B 0.000,C 90.000,E1 81.837} C_DIS
LIN {X 0.016,Y -581.829,Z 1365.246,A 0.000,B 0.000,C 90.000,E1 80.208} C_DIS
LIN {X 0.273,Y -583.045,Z 1365.240,A 0.000,B 0.000,C 90.000,E1 79.106} C_DIS
LIN {X 0.083,Y -584.087,Z 1365.234,A 0.000,B 0.000,C 90.000,E1 78.049} C_DIS
LIN {X 0.154,Y -585.375,Z 1365.226,A 0.000,B 0.000,C 90.000,E1 76.700} C_DIS
LIN {X -0.007,Y -586.218,Z 1365.220,A 0.000,B 0.000,C 90.000,E1 75.644} C_DIS
LIN {X 0.228,Y -587.178,Z 1365.213,A 0.000,B 0.000,C 90.000,E1 74.283} C_DIS
LIN {X 0.173,Y -588.365,Z 1365.203,A 0.000,B 0.000,C 90.000,E1 72.417} C_DIS
LIN {X 0.185,Y -588.987,Z 1365.197,A 0.000,B 0.000,C 90.000,E1 71.348} C_DIS
LIN {X -0.196,Y -590.030,Z 1365.186,A 0.000,B 0.000,C 90.000,E1 69.518} C_DIS
LIN {X -0.224,Y -591.014,Z 1365.177,A 0.000,B 0.000,C 90.000,E1 67.922} C_DIS
LIN {X -0.113,Y -592.384,Z 1365.167,A 0.000,B 0.000,C 90.000,E1 66.049} C_DIS
LIN {X -0.161,Y -593.741,Z 1365.158,A 0.000,B 0.000,C 90.000,E1 64.460} C_DIS
LIN {X -0.180,Y -594.893,Z 1365.149,A 0.000,B 0.000,C 90.000,E1 62.871} C_DIS
LIN {X -0.001,Y -596.374,Z 1365.139,A 0.000,B 0.000,C 90.000,E1 61.001} C_DIS
LIN {X 0.151,Y -597.626,Z 1365.132,A 0.000,B 0.000,C 90.000,E1 59.665} C_DIS
LIN {X -0.267,Y -599.147,Z 1365.123,A 0.000,B 0.000,C 90.000,E1 58.122} C_DIS
LIN {X 0.022,Y -600.163,Z 1365.117,A 0.000,B 0.000,C 90.000,E1 57.041} C_DIS
LIN {X 0.065,Y -601.391,Z 1365.110,A 0.000,B 0.000,C 90.000,E1 55.722} C_DIS
LIN {X 0.031,Y -602.853,Z 1365.101,A 0.000,B 0.000,C 90.000,E1 54.149} C_DIS
LIN {X 0.238,Y -604.303,Z 1365.092,A 0.000,B 0.000,C 90.000,E1 52.557} C_DIS
LIN {X -0.045,Y -605.097,Z 1365.086,A 0.000,B 0.000,C 90.000,E1 51.537} C_DIS
LIN {X -0.060,Y -605.855,Z 1365.079,A 0.000,B 0.000,C 90.000,E1 50.231} C_DIS
LIN {X 0.058,Y -606.439,Z 1365.073,A 0.000,B 0.000,C 90.000,E1 49.175} C_DIS
LIN {X -0.271,Y -606.824,Z 1365.068,A 0.000,B 0.000,C 90.000,E1 48.162} C_DIS
LIN {X 0.081,Y -607.144,Z 1365.060,A 0.000,B 0.000,C 90.000,E1 46.824} C_DIS
LIN {X 0.012,Y -607.261,Z 1365.053,A 0.000,B 0.000,C 90.000,E1 45.526} C_DIS
LIN {X 0.359,Y -607.118,Z 1365.046,A 0.000,B 0.000,C 90.000,E1 44.190} C_DIS
LIN {X 0.043,Y -606.749,Z 1365.040,A 0.000,B 0.000,C 90.000,E1 43.176} C_DIS
LIN {X -0.062,Y -606.144,Z 1365.033,A 0.000,B 0.000,C 90.000,E1 41.881} C_DIS
LIN {X 0.056,Y -605.636,Z 1365.027,A 0.000,B 0.000,C 90.000,E1 40.825} C_DIS
LIN {X -0.165,Y -604.612,Z 1365.018,A 0.000,B 0.000,C 90.000,E1 39.277} C_DIS
LIN {X 0.188,Y -603.588,Z 1365.011,A 0.000,B 0.000,C 90.000,E1 37.935} C_DIS
LIN {X 0.370,Y -602.599,Z 1365.005,A 0.000,B 0.000,C 90.000,E1 36.870} C_DIS
LIN {X 0.289,Y -601.670,Z 1365.001,A 0.000,B 0.000,C 90.000,E1 36.091} C_DIS
LIN {X -0.148,Y -599.517,Z 1364.993,A 0.000,B 0.000,C 90.000,E1 34.818} C_DIS
LIN {X -0.133,Y -596.706,Z 1364.986,A 0.000,B 0.000,C 90.000,E1 33.499} C_DIS
LIN {X 0.111,Y -594.150,Z 1364.980,A 0.000,B 0.000,C 90.000,E1 32.418} C_DIS
LIN {X 0.118,Y -591.916,Z 1364.976,A 0.000,B 0.000,C 90.000,E1 31.623} C_DIS
LIN {X -0.097,Y -589.371,Z 1364.971,A 0.000,B 0.000,C 90.000,E1 30.846} C_DIS
LIN {X -0.263,Y -585.431,Z 1364.965,A 0.000,B 0.000,C 90.000,E1 29.795} C_DIS
LIN {X 0.162,Y -582.143,Z 1364.961,A 0.000,B 0.000,C 90.000,E1 28.949} C_DIS
LIN {X -0.033,Y -580.283,Z 1364.959,A 0.000,B 0.000,C 90.000,E1 28.565} C_DIS
LIN {X -0.250,Y -575.653,Z 1364.953,A 0.000,B 0.000,C 90.000,E1 27.641} C_DIS
LIN {X 0.057,Y -571.277,Z 1364.949,A 0.000,B 0.000,C 90.000,E1 26.796} C_DIS
LIN {X 0.233,Y -568.167,Z 1364.946,A 0.000,B 0.000,C 90.000,E1 26.232} C_DIS
LIN {X -0.211,Y -563.962,Z 1364.942,A 0.000,B 0.000,C 90.000,E1 25.591} C_DIS
LIN {X -0.180,Y -559.497,Z 1364.938,A 0.000,B 0.000,C 90.000,E1 24.899} C_DIS
LIN {X -0.188,Y -554.593,Z 1364.934,A 0.000,B 0.000,C 90.000,E1 24.207} C_DIS
LIN {X 0.148,Y -548.269,Z 1364.930,A 0.000,B 0.000,C 90.000,E1 23.334} C_DIS
LIN {X -0.092,Y -541.381,Z 1364.925,A 0.000,B 0.000,C 90.000,E1 22.514} C_DIS
LIN {X 0.231,Y -535.311,Z 1364.921,A 0.000,B 0.000,C 90.000,E1 21.770} C_DIS
LIN {X -0.136,Y -527.672,Z 1364.917,A 0.000,B 0.000,C 90.000,E1 20.972} C_DIS
LIN {X 0.116,Y -522.381,Z 1364.913,A 0.000,B 0.000,C 90.000,E1 20.375} C_DIS
LIN {X 0.205,Y -513.136,Z 1364.908,A 0.000,B 0.000,C 90.000,E1 19.396} C_DIS
LIN {X -0.264,Y -502.676,Z 1364.902,A 0.000,B 0.000,C 90.000,E1 18.362} C_DIS
LIN {X 0.166,Y -493.288,Z 1364.896,A 0.000,B 0.000,C 90.000,E1 17.347} C_DIS
LIN {X 0.169,Y -482.105,Z 1364.891,A 0.000,B 0.000,C 90.000,E1 16.260} C_DIS
LIN {X -0.232,Y -466.626,Z 1364.882,A 0.000,B 0.000,C 90.000,E1 14.773} C_DIS
LIN {X 0.141,Y -455.224,Z 1364.876,A 0.000,B 0.000,C 90.000,E1 13.592} C_DIS
LIN {X 0.187,Y -438.163,Z 1364.866,A 0.000,B 0.000,C 90.000,E1 11.827} C_DIS
LIN {X 0.039,Y -424.173,Z 1364.857,A 0.000,B 0.000,C 90.000,E1 10.310} C_DIS
LIN {X -0.196,Y -411.679,Z 1364.849,A 0.000,B 0.000,C 90.000,E1 8.916} C_DIS
LIN {X -0.104,Y -401.841,Z 1364.843,A 0.000,B 0.000,C 90.000,E1 7.757} C_DIS
LIN {X 0.138,Y -397.656,Z 1364.840,A 0.000,B 0.000,C 90.000,E1 7.239} C_DIS
LIN {X 0.089,Y -392.803,Z 1364.837,A 0.000,B 0.000,C 90.000,E1 6.549} C_DIS
LIN {X 0.051,Y -392.790,Z 1364.836,A 0.000,B 0.000,C 90.000,E1 6.549} C_DIS
LIN {X -0.050,Y -394.263,Z 1364.835,A 0.000,B 0.000,C 90.000,E1 6.315} C_DIS
LIN {X 0.121,Y -397.789,Z 1364.833,A 0.000,B 0.000,C 90.000,E1 5.967} C_DIS
LIN {X -0.187,Y -402.133,Z 1364.831,A 0.000,B 0.000,C 90.000,E1 5.682} C_DIS
LIN {X 0.149,Y -410.332,Z 1364.828,A 0.000,B 0.000,C 90.000,E1 5.049} C_DIS
LIN {X -0.177,Y -416.495,Z 1364.825,A 0.000,B 0.000,C 90.000,E1 4.588} C_DIS
LIN {X 0.210,Y -423.813,Z 1364.822,A 0.000,B 0.000,C 90.000,E1 3.841} C_DIS
LIN {X 0.086,Y -430.592,Z 1364.817,A 0.000,B 0.000,C 90.000,E1 3.094} C_DIS
LIN {X 0.035,Y -437.235,Z 1364.813,A 0.000,B 0.000,C 90.000,E1 2.293} C_DIS
LIN {X -0.124,Y -443.668,Z 1364.808,A 0.000,B 0.000,C 90.000,E1 1.489} C_DIS
LIN {X 0.138,Y -448.529,Z 1364.805,A 0.000,B 0.000,C 90.000,E1 0.802} C_DIS
LIN {X -0.006,Y -453.234,Z 1364.801,A 0.000,B 0.000,C 90.000,E1 0.172} C_DIS
LIN {X 0.082,Y -459.965,Z 1364.795,A 0.000,B 0.000,C 90.000,E1 359.141} C_DIS
LIN {X 0.022,Y -464.004,Z 1364.792,A 0.000,B 0.000,C 90.000,E1 358.511} C_DIS
LIN {X -0.232,Y -469.491,Z 1364.786,A 0.000,B 0.000,C 90.000,E1 357.593} C_DIS
LIN {X -0.225,Y -472.943,Z 1364.783,A 0.000,B 0.000,C 90.000,E1 356.963} C_DIS
LIN {X -0.037,Y -476.921,Z 1364.779,A 0.000,B 0.000,C 90.000,E1 356.159} C_DIS
LIN {X 0.192,Y -480.559,Z 1364.774,A 0.000,B 0.000,C 90.000,E1 355.355} C_DIS
LIN {X -0.167,Y -483.268,Z 1364.771,A 0.000,B 0.000,C 90.000,E1 354.780} C_DIS
LIN {X -0.024,Y -485.798,Z 1364.767,A 0.000,B 0.000,C 90.000,E1 354.147} C_DIS
LIN {X 0.006,Y -489.203,Z 1364.762,A 0.000,B 0.000,C 90.000,E1 353.223} C_DIS
LIN {X 0.075,Y -492.317,Z 1364.757,A 0.000,B 0.000,C 90.000,E1 352.299} C_DIS
LIN {X 0.177,Y -495.070,Z 1364.752,A 0.000,B 0.000,C 90.000,E1 351.376} C_DIS
LIN {X -0.103,Y -497.465,Z 1364.747,A 0.000,B 0.000,C 90.000,E1 350.500} C_DIS
LIN {X 0.050,Y -499.644,Z 1364.742,A 0.000,B 0.000,C 90.000,E1 349.577} C_DIS
LIN {X -0.179,Y -501.618,Z 1364.737,A 0.000,B 0.000,C 90.000,E1 348.701} C_DIS
LIN {X 0.212,Y -503.393,Z 1364.732,A 0.000,B 0.000,C 90.000,E1 347.757} C_DIS
LIN {X -0.034,Y -505.434,Z 1364.725,A 0.000,B 0.000,C 90.000,E1 346.589} C_DIS
LIN {X -0.084,Y -506.821,Z 1364.721,A 0.000,B 0.000,C 90.000,E1 345.700} C_DIS
LIN {X -0.063,Y -507.510,Z 1364.717,A 0.000,B 0.000,C 90.000,E1 345.102} C_DIS
LIN {X -0.116,Y -507.726,Z 1364.716,A 0.000,B 0.000,C 90.000,E1 344.810} C_DIS
LIN {X -0.169,Y -507.763,Z 1364.714,A 0.000,B 0.000,C 90.000,E1 344.519} C_DIS
LIN {X -0.086,Y -507.617,Z 1364.712,A 0.000,B 0.000,C 90.000,E1 344.212} C_DIS
LIN {X -0.140,Y -507.130,Z 1364.711,A 0.000,B 0.000,C 90.000,E1 343.921} C_DIS
LIN {X -0.053,Y -506.048,Z 1364.709,A 0.000,B 0.000,C 90.000,E1 343.614} C_DIS
LIN {X 0.089,Y -504.786,Z 1364.708,A 0.000,B 0.000,C 90.000,E1 343.449} C_DIS
LIN {X -0.110,Y -500.730,Z 1364.707,A 0.000,B 0.000,C 90.000,E1 343.323} C_DIS
LIN {X 0.013,Y -469.460,Z 1364.701,A 0.000,B 0.000,C 90.000,E1 342.181} C_DIS
LIN {X -0.101,Y -438.437,Z 1364.694,A 0.000,B 0.000,C 90.000,E1 340.913} C_DIS
LIN {X 0.216,Y -411.100,Z 1364.687,A 0.000,B 0.000,C 90.000,E1 339.571} C_DIS
LIN {X -0.079,Y -385.646,Z 1364.679,A 0.000,B 0.000,C 90.000,E1 338.230} C_DIS
LIN {X -0.059,Y -362.529,Z 1364.671,A 0.000,B 0.000,C 90.000,E1 336.794} C_DIS
LIN {X -0.081,Y -362.519,Z 1364.671,A 0.000,B 0.000,C 90.000,E1 336.794} C_DIS
LIN {X -0.056,Y -366.191,Z 1364.641,A 0.000,B 0.000,C 90.000,E1 331.435} C_DIS
LIN {X -0.031,Y -371.208,Z 1364.604,A 0.000,B 0.000,C 90.000,E1 324.769} C_DIS
LIN {X -0.044,Y -371.641,Z 1364.602,A 0.000,B 0.000,C 90.000,E1 324.402} C_DIS
LIN {X 0.012,Y -376.746,Z 1364.570,A 0.000,B 0.000,C 90.000,E1 318.528} C_DIS
LIN {X -0.232,Y -378.141,Z 1364.564,A 0.000,B 0.000,C 90.000,E1 317.472} C_DIS
LIN {X 0.041,Y -384.262,Z 1364.529,A 0.000,B 0.000,C 90.000,E1 311.272} C_DIS
LIN {X 0.084,Y -384.767,Z 1364.527,A 0.000,B 0.000,C 90.000,E1 310.906} C_DIS
LIN {X 0.074,Y -390.932,Z 1364.494,A 0.000,B 0.000,C 90.000,E1 304.818} C_DIS
LIN {X -0.081,Y -391.358,Z 1364.492,A 0.000,B 0.000,C 90.000,E1 304.485} C_DIS
LIN {X 0.090,Y -397.066,Z 1364.458,A 0.000,B 0.000,C 90.000,E1 298.437} C_DIS
LIN {X 0.046,Y -401.470,Z 1364.427,A 0.000,B 0.000,C 90.000,E1 292.823} C_DIS
LIN {X 0.128,Y -401.680,Z 1364.425,A 0.000,B 0.000,C 90.000,E1 292.461} C_DIS
LIN {X 0.173,Y -404.553,Z 1364.396,A 0.000,B 0.000,C 90.000,E1 287.221} C_DIS
LIN {X -0.113,Y -404.761,Z 1364.394,A 0.000,B 0.000,C 90.000,E1 286.913} C_DIS
LIN {X -0.216,Y -406.030,Z 1364.365,A 0.000,B 0.000,C 90.000,E1 281.715} C_DIS
LIN {X -0.207,Y -406.144,Z 1364.363,A 0.000,B 0.000,C 90.000,E1 281.366} C_DIS
LIN {X -0.102,Y -405.651,Z 1364.334,A 0.000,B 0.000,C 90.000,E1 276.144} C_DIS
LIN {X -0.098,Y -405.612,Z 1364.332,A 0.000,B 0.000,C 90.000,E1 275.796} C_DIS
LIN {X -0.025,Y -403.552,Z 1364.305,A 0.000,B 0.000,C 90.000,E1 270.917} C_DIS
LIN {X -0.089,Y -403.057,Z 1364.301,A 0.000,B 0.000,C 90.000,E1 270.229} C_DIS
LIN {X 0.135,Y -399.016,Z 1364.272,A 0.000,B 0.000,C 90.000,E1 264.951} C_DIS
LIN {X 0.029,Y -397.652,Z 1364.266,A 0.000,B 0.000,C 90.000,E1 263.913} C_DIS
LIN {X -0.090,Y -392.934,Z 1364.241,A 0.000,B 0.000,C 90.000,E1 259.342} C_DIS
LIN {X -0.133,Y -392.480,Z 1364.239,A 0.000,B 0.000,C 90.000,E1 258.993} C_DIS
LIN {X 0.016,Y -386.124,Z 1364.213,A 0.000,B 0.000,C 90.000,E1 254.338} C_DIS
LIN {X -0.024,Y -384.993,Z 1364.207,A 0.000,B 0.000,C 90.000,E1 253.268} C_DIS
LIN {X -0.150,Y -378.134,Z 1364.183,A 0.000,B 0.000,C 90.000,E1 248.954} C_DIS
LIN {X 0.064,Y -375.883,Z 1364.173,A 0.000,B 0.000,C 90.000,E1 247.102} C_DIS
LIN {X 0.013,Y -369.105,Z 1364.151,A 0.000,B 0.000,C 90.000,E1 243.076} C_DIS
LIN {X 0.092,Y -366.258,Z 1364.138,A 0.000,B 0.000,C 90.000,E1 240.845} C_DIS
LIN {X 0.053,Y -358.852,Z 1364.113,A 0.000,B 0.000,C 90.000,E1 236.373} C_DIS
LIN {X 0.041,Y -356.042,Z 1364.101,A 0.000,B 0.000,C 90.000,E1 234.116} C_DIS
LIN {X 0.037,Y -348.479,Z 1364.073,A 0.000,B 0.000,C 90.000,E1 229.175} C_DIS
LIN {X 0.098,Y -345.899,Z 1364.061,A 0.000,B 0.000,C 90.000,E1 226.863} C_DIS
LIN {X 0.064,Y -339.124,Z 1364.033,A 0.000,B 0.000,C 90.000,E1 221.838} C_DIS
LIN {X 0.149,Y -336.957,Z 1364.020,A 0.000,B 0.000,C 90.000,E1 219.483} C_DIS
LIN {X -0.151,Y -333.591,Z 1364.004,A 0.000,B 0.000,C 90.000,E1 216.790} C_DIS
LIN {X 0.026,Y -329.370,Z 1363.976,A 0.000,B 0.000,C 90.000,E1 211.623} C_DIS
LIN {X -0.072,Y -328.648,Z 1363.971,A 0.000,B 0.000,C 90.000,E1 210.846} C_DIS
LIN {X 0.038,Y -325.151,Z 1363.947,A 0.000,B 0.000,C 90.000,E1 206.437} C_DIS
LIN {X 0.021,Y -325.167,Z 1363.947,A 0.000,B 0.000,C 90.000,E1 206.437} C_DIS
LIN {X 0.064,Y -345.062,Z 1363.938,A 0.000,B 0.000,C 90.000,E1 204.847} C_DIS
LIN {X 0.212,Y -365.559,Z 1363.930,A 0.000,B 0.000,C 90.000,E1 203.387} C_DIS
LIN {X 0.037,Y -387.994,Z 1363.922,A 0.000,B 0.000,C 90.000,E1 202.025} C_DIS
LIN {X 0.124,Y -412.361,Z 1363.915,A 0.000,B 0.000,C 90.000,E1 200.684} C_DIS
LIN {X 0.135,Y -440.436,Z 1363.908,A 0.000,B 0.000,C 90.000,E1 199.341} C_DIS
LIN {X -0.086,Y -443.961,Z 1363.907,A 0.000,B 0.000,C 90.000,E1 199.214} C_DIS
LIN {X 0.128,Y -447.067,Z 1363.906,A 0.000,B 0.000,C 90.000,E1 199.033} C_DIS
LIN {X -0.210,Y -448.409,Z 1363.905,A 0.000,B 0.000,C 90.000,E1 198.906} C_DIS
LIN {X -0.065,Y -449.216,Z 1363.904,A 0.000,B 0.000,C 90.000,E1 198.725} C_DIS
LIN {X 0.083,Y -449.815,Z 1363.903,A 0.000,B 0.000,C 90.000,E1 198.544} C_DIS
LIN {X -0.043,Y -450.706,Z 1363.901,A 0.000,B 0.000,C 90.000,E1 198.236} C_DIS
LIN {X 0.261,Y -451.350,Z 1363.900,A 0.000,B 0.000,C 90.000,E1 197.873} C_DIS
LIN {X -0.119,Y -452.179,Z 1363.896,A 0.000,B 0.000,C 90.000,E1 197.275} C_DIS
LIN {X -0.109,Y -453.362,Z 1363.887,A 0.000,B 0.000,C 90.000,E1 195.662} C_DIS
LIN {X 0.039,Y -454.276,Z 1363.880,A 0.000,B 0.000,C 90.000,E1 194.356} C_DIS
LIN {X -0.139,Y -455.291,Z 1363.871,A 0.000,B 0.000,C 90.000,E1 192.771} C_DIS
LIN {X -0.068,Y -456.077,Z 1363.864,A 0.000,B 0.000,C 90.000,E1 191.478} C_DIS
LIN {X 0.150,Y -456.969,Z 1363.855,A 0.000,B 0.000,C 90.000,E1 189.849} C_DIS
LIN {X 0.153,Y -457.438,Z 1363.848,A 0.000,B 0.000,C 90.000,E1 188.568} C_DIS
LIN {X 0.092,Y -457.802,Z 1363.841,A 0.000,B 0.000,C 90.000,E1 187.296} C_DIS
LIN {X 0.210,Y -458.171,Z 1363.832,A 0.000,B 0.000,C 90.000,E1 185.682} C_DIS
LIN {X 0.160,Y -458.317,Z 1363.828,A 0.000,B 0.000,C 90.000,E1 185.049} C_DIS
LIN {X -0.211,Y -458.120,Z 1363.819,A 0.000,B 0.000,C 90.000,E1 183.498} C_DIS
LIN {X -0.075,Y -457.940,Z 1363.814,A 0.000,B 0.000,C 90.000,E1 182.522} C_DIS
LIN {X -0.214,Y -457.415,Z 1363.807,A 0.000,B 0.000,C 90.000,E1 181.260} C_DIS
LIN {X -0.102,Y -456.657,Z 1363.802,A 0.000,B 0.000,C 90.000,E1 180.286} C_DIS
LIN {X -0.184,Y -456.017,Z 1363.798,A 0.000,B 0.000,C 90.000,E1 179.656} C_DIS
LIN {X -0.176,Y -453.275,Z 1363.789,A 0.000,B 0.000,C 90.000,E1 178.051} C_DIS
LIN {X -0.119,Y -451.080,Z 1363.784,A 0.000,B 0.000,C 90.000,E1 177.078} C_DIS
LIN {X 0.225,Y -449.270,Z 1363.780,A 0.000,B 0.000,C 90.000,E1 176.388} C_DIS
LIN {X -0.193,Y -445.962,Z 1363.775,A 0.000,B 0.000,C 90.000,E1 175.469} C_DIS
LIN {X 0.109,Y -443.297,Z 1363.771,A 0.000,B 0.000,C 90.000,E1 174.780} C_DIS
LIN {X 0.097,Y -438.706,Z 1363.766,A 0.000,B 0.000,C 90.000,E1 173.799} C_DIS
LIN {X 0.032,Y -433.091,Z 1363.760,A 0.000,B 0.000,C 90.000,E1 172.818} C_DIS
LIN {X -0.101,Y -426.609,Z 1363.755,A 0.000,B 0.000,C 90.000,E1 171.837} C_DIS
LIN {X -0.108,Y -415.017,Z 1363.745,A 0.000,B 0.000,C 90.000,E1 170.151} C_DIS
LIN {X 0.045,Y -405.909,Z 1363.738,A 0.000,B 0.000,C 90.000,E1 168.757} C_DIS
LIN {X 0.186,Y -395.307,Z 1363.728,A 0.000,B 0.000,C 90.000,E1 166.992} C_DIS
LIN {X 0.109,Y -391.730,Z 1363.724,A 0.000,B 0.000,C 90.000,E1 166.297} C_DIS
LIN {X -0.147,Y -390.649,Z 1363.722,A 0.000,B 0.000,C 90.000,E1 166.047} C_DIS
LIN {X 0.196,Y -389.256,Z 1363.719,A 0.000,B 0.000,C 90.000,E1 165.463} C_DIS
LIN {X 0.215,Y -389.089,Z 1363.719,A 0.000,B 0.000,C 90.000,E1 165.283} C_DIS
LIN {X -0.075,Y -389.182,Z 1363.718,A 0.000,B 0.000,C 90.000,E1 165.172} C_DIS
LIN {X 0.083,Y -389.626,Z 1363.717,A 0.000,B 0.000,C 90.000,E1 165.046} C_DIS
LIN {X 0.031,Y -392.477,Z 1363.715,A 0.000,B 0.000,C 90.000,E1 164.629} C_DIS
LIN {X 0.032,Y -399.669,Z 1363.710,A 0.000,B 0.000,C 90.000,E1 163.795} C_DIS
LIN {X 0.172,Y -406.589,Z 1363.706,A 0.000,B 0.000,C 90.000,E1 163.087} C_DIS
LIN {X -0.024,Y -420.686,Z 1363.699,A 0.000,B 0.000,C 90.000,E1 161.873} C_DIS
LIN {X -0.167,Y -446.137,Z 1363.688,A 0.000,B 0.000,C 90.000,E1 159.880} C_DIS
LIN {X 0.072,Y -457.072,Z 1363.684,A 0.000,B 0.000,C 90.000,E1 159.028} C_DIS
LIN {X 0.238,Y -466.132,Z 1363.680,A 0.000,B 0.000,C 90.000,E1 158.284} C_DIS
LIN {X 0.148,Y -472.122,Z 1363.677,A 0.000,B 0.000,C 90.000,E1 157.794} C_DIS
LIN {X -0.105,Y -479.567,Z 1363.673,A 0.000,B 0.000,C 90.000,E1 157.177} C_DIS
LIN {X 0.215,Y -485.357,Z 1363.670,A 0.000,B 0.000,C 90.000,E1 156.613} C_DIS
LIN {X -0.153,Y -493.916,Z 1363.666,A 0.000,B 0.000,C 90.000,E1 155.845} C_DIS
LIN {X -0.092,Y -500.707,Z 1363.662,A 0.000,B 0.000,C 90.000,E1 155.153} C_DIS
LIN {X 0.208,Y -504.588,Z 1363.660,A 0.000,B 0.000,C 90.000,E1 154.717} C_DIS
LIN {X 0.164,Y -510.765,Z 1363.656,A 0.000,B 0.000,C 90.000,E1 154.024} C_DIS
LIN {X -0.087,Y -515.805,Z 1363.653,A 0.000,B 0.000,C 90.000,E1 153.461} C_DIS
LIN {X 0.093,Y -519.346,Z 1363.650,A 0.000,B 0.000,C 90.000,E1 152.999} C_DIS
LIN {X 0.137,Y -523.733,Z 1363.647,A 0.000,B 0.000,C 90.000,E1 152.410} C_DIS
LIN {X 0.122,Y -526.801,Z 1363.644,A 0.000,B 0.000,C 90.000,E1 151.975} C_DIS
LIN {X 0.221,Y -530.487,Z 1363.641,A 0.000,B 0.000,C 90.000,E1 151.385} C_DIS
LIN {X -0.117,Y -533.531,Z 1363.638,A 0.000,B 0.000,C 90.000,E1 150.845} C_DIS
LIN {X -0.107,Y -536.823,Z 1363.634,A 0.000,B 0.000,C 90.000,E1 150.127} C_DIS
LIN {X -0.075,Y -539.671,Z 1363.630,A 0.000,B 0.000,C 90.000,E1 149.410} C_DIS
LIN {X 0.113,Y -541.633,Z 1363.627,A 0.000,B 0.000,C 90.000,E1 148.820} C_DIS
LIN {X 0.137,Y -543.400,Z 1363.624,A 0.000,B 0.000,C 90.000,E1 148.250} C_DIS
LIN {X 0.086,Y -545.629,Z 1363.619,A 0.000,B 0.000,C 90.000,E1 147.406} C_DIS
LIN {X -0.114,Y -547.383,Z 1363.614,A 0.000,B 0.000,C 90.000,E1 146.580} C_DIS
LIN {X -0.249,Y -549.367,Z 1363.608,A 0.000,B 0.000,C 90.000,E1 145.468} C_DIS
LIN {X -0.093,Y -550.541,Z 1363.603,A 0.000,B 0.000,C 90.000,E1 144.609} C_DIS
LIN {X -0.242,Y -551.521,Z 1363.599,A 0.000,B 0.000,C 90.000,E1 143.783} C_DIS
LIN {X -0.059,Y -552.311,Z 1363.594,A 0.000,B 0.000,C 90.000,E1 142.924} C_DIS
LIN {X -0.238,Y -553.205,Z 1363.588,A 0.000,B 0.000,C 90.000,E1 141.823} C_DIS
LIN {X 0.087,Y -554.308,Z 1363.578,A 0.000,B 0.000,C 90.000,E1 140.114} C_DIS
LIN {X 0.016,Y -555.334,Z 1363.569,A 0.000,B 0.000,C 90.000,E1 138.447} C_DIS
LIN {X -0.047,Y -556.138,Z 1363.560,A 0.000,B 0.000,C 90.000,E1 136.782} C_DIS
LIN {X -0.187,Y -556.730,Z 1363.552,A 0.000,B 0.000,C 90.000,E1 135.405} C_DIS
LIN {X 0.135,Y -557.424,Z 1363.543,A 0.000,B 0.000,C 90.000,E1 133.704} C_DIS
LIN {X -0.187,Y -558.814,Z 1363.531,A 0.000,B 0.000,C 90.000,E1 131.515} C_DIS
LIN {X 0.113,Y -559.724,Z 1363.527,A 0.000,B 0.000,C 90.000,E1 130.825} C_DIS
LIN {X -0.056,Y -559.784,Z 1363.527,A 0.000,B 0.000,C 90.000,E1 130.825} C_DIS
LIN {X -0.098,Y -559.800,Z 1363.527,A 0.000,B 0.000,C 90.000,E1 130.825} C_DIS
LIN {X 0.047,Y -562.952,Z 1363.525,A 0.000,B 0.000,C 90.000,E1 130.539} C_DIS
LIN {X -0.198,Y -567.986,Z 1363.524,A 0.000,B 0.000,C 90.000,E1 130.378} C_DIS
LIN {X -0.107,Y -577.091,Z 1363.523,A 0.000,B 0.000,C 90.000,E1 130.092} C_DIS
LIN {X 0.072,Y -580.201,Z 1363.522,A 0.000,B 0.000,C 90.000,E1 129.967} C_DIS
LIN {X -0.189,Y -585.982,Z 1363.521,A 0.000,B 0.000,C 90.000,E1 129.725} C_DIS
LIN {X 0.042,Y -591.758,Z 1363.519,A 0.000,B 0.000,C 90.000,E1 129.358} C_DIS
LIN {X 0.112,Y -597.552,Z 1363.516,A 0.000,B 0.000,C 90.000,E1 128.955} C_DIS
LIN {X -0.078,Y -603.085,Z 1363.514,A 0.000,B 0.000,C 90.000,E1 128.543} C_DIS
LIN {X -0.185,Y -608.383,Z 1363.512,A 0.000,B 0.000,C 90.000,E1 128.096} C_DIS
LIN {X -0.026,Y -613.603,Z 1363.509,A 0.000,B 0.000,C 90.000,E1 127.604} C_DIS
LIN {X 0.001,Y -617.392,Z 1363.507,A 0.000,B 0.000,C 90.000,E1 127.237} C_DIS
LIN {X 0.264,Y -623.378,Z 1363.503,A 0.000,B 0.000,C 90.000,E1 126.583} C_DIS
LIN {X -0.091,Y -630.359,Z 1363.499,A 0.000,B 0.000,C 90.000,E1 125.851} C_DIS
LIN {X 0.268,Y -634.704,Z 1363.496,A 0.000,B 0.000,C 90.000,E1 125.311} C_DIS
LIN {X 0.139,Y -638.758,Z 1363.494,A 0.000,B 0.000,C 90.000,E1 124.818} C_DIS
LIN {X -0.431,Y -645.415,Z 1363.489,A 0.000,B 0.000,C 90.000,E1 123.992} C_DIS
LIN {X 0.437,Y -649.804,Z 1363.485,A 0.000,B 0.000,C 90.000,E1 123.293} C_DIS
LIN {X 0.047,Y -653.100,Z 1363.482,A 0.000,B 0.000,C 90.000,E1 122.832} C_DIS
LIN {X 0.031,Y -656.065,Z 1363.480,A 0.000,B 0.000,C 90.000,E1 122.339} C_DIS
LIN {X -0.319,Y -658.765,Z 1363.477,A 0.000,B 0.000,C 90.000,E1 121.878} C_DIS
LIN {X -0.186,Y -662.346,Z 1363.473,A 0.000,B 0.000,C 90.000,E1 121.131} C_DIS
LIN {X 0.412,Y -664.441,Z 1363.470,A 0.000,B 0.000,C 90.000,E1 120.590} C_DIS
LIN {X 0.259,Y -666.993,Z 1363.466,A 0.000,B 0.000,C 90.000,E1 119.873} C_DIS
LIN {X 0.134,Y -669.083,Z 1363.462,A 0.000,B 0.000,C 90.000,E1 119.155} C_DIS
LIN {X -0.292,Y -669.729,Z 1363.461,A 0.000,B 0.000,C 90.000,E1 118.949} C_DIS
LIN {X -0.393,Y -670.869,Z 1363.457,A 0.000,B 0.000,C 90.000,E1 118.231} C_DIS
LIN {X -0.058,Y -671.227,Z 1363.454,A 0.000,B 0.000,C 90.000,E1 117.719} C_DIS
LIN {X -0.314,Y -671.327,Z 1363.451,A 0.000,B 0.000,C 90.000,E1 117.257} C_DIS
LIN {X 0.198,Y -671.205,Z 1363.447,A 0.000,B 0.000,C 90.000,E1 116.488} C_DIS
LIN {X -0.190,Y -670.781,Z 1363.443,A 0.000,B 0.000,C 90.000,E1 115.796} C_DIS
LIN {X 0.148,Y -670.351,Z 1363.441,A 0.000,B 0.000,C 90.000,E1 115.283} C_DIS
LIN {X -0.127,Y -669.690,Z 1363.438,A 0.000,B 0.000,C 90.000,E1 114.823} C_DIS
LIN {X -0.243,Y -669.180,Z 1363.437,A 0.000,B 0.000,C 90.000,E1 114.591} C_DIS
LIN {X 0.080,Y -667.706,Z 1363.434,A 0.000,B 0.000,C 90.000,E1 114.079} C_DIS
LIN {X 0.194,Y -663.950,Z 1363.431,A 0.000,B 0.000,C 90.000,E1 113.462} C_DIS
LIN {X 0.266,Y -662.764,Z 1363.430,A 0.000,B 0.000,C 90.000,E1 113.334} C_DIS
LIN {X -0.220,Y -657.268,Z 1363.427,A 0.000,B 0.000,C 90.000,E1 112.950} C_DIS
LIN {X -0.003,Y -655.340,Z 1363.427,A 0.000,B 0.000,C 90.000,E1 112.823} C_DIS
LIN {X -0.117,Y -649.219,Z 1363.426,A 0.000,B 0.000,C 90.000,E1 112.589} C_DIS
LIN {X -0.114,Y -645.127,Z 1363.425,A 0.000,B 0.000,C 90.000,E1 112.461} C_DIS
LIN {X -0.038,Y -637.338,Z 1363.424,A 0.000,B 0.000,C 90.000,E1 112.259} C_DIS
LIN {X 0.109,Y -630.693,Z 1363.423,A 0.000,B 0.000,C 90.000,E1 112.078} C_DIS
LIN {X 0.049,Y -630.532,Z 1363.423,A 0.000,B 0.000,C 90.000,E1 112.078} C_DIS
LIN {X -0.256,Y -630.990,Z 1363.422,A 0.000,B 0.000,C 90.000,E1 112.025} C_DIS
LIN {X -0.012,Y -640.316,Z 1363.416,A 0.000,B 0.000,C 90.000,E1 110.918} C_DIS
LIN {X -0.143,Y -644.428,Z 1363.413,A 0.000,B 0.000,C 90.000,E1 110.429} C_DIS
LIN {X -0.215,Y -648.571,Z 1363.410,A 0.000,B 0.000,C 90.000,E1 109.812} C_DIS
LIN {X 0.219,Y -653.378,Z 1363.405,A 0.000,B 0.000,C 90.000,E1 108.906} C_DIS
LIN {X -0.075,Y -657.939,Z 1363.400,A 0.000,B 0.000,C 90.000,E1 107.946} C_DIS
LIN {X -0.208,Y -661.095,Z 1363.396,A 0.000,B 0.000,C 90.000,E1 107.221} C_DIS
LIN {X -0.218,Y -663.041,Z 1363.393,A 0.000,B 0.000,C 90.000,E1 106.732} C_DIS
LIN {X 0.230,Y -664.837,Z 1363.390,A 0.000,B 0.000,C 90.000,E1 106.205} C_DIS
LIN {X 0.238,Y -666.417,Z 1363.387,A 0.000,B 0.000,C 90.000,E1 105.717} C_DIS
LIN {X -0.005,Y -668.356,Z 1363.383,A 0.000,B 0.000,C 90.000,E1 105.009} C_DIS
LIN {X -0.226,Y -669.732,Z 1363.379,A 0.000,B 0.000,C 90.000,E1 104.300} C_DIS
LIN {X 0.285,Y -670.433,Z 1363.377,A 0.000,B 0.000,C 90.000,E1 103.772} C_DIS
LIN {X 0.151,Y -670.897,Z 1363.374,A 0.000,B 0.000,C 90.000,E1 103.300} C_DIS
LIN {X -0.046,Y -671.162,Z 1363.370,A 0.000,B 0.000,C 90.000,E1 102.591} C_DIS
LIN {X -0.179,Y -671.167,Z 1363.367,A 0.000,B 0.000,C 90.000,E1 102.119} C_DIS
LIN {X 0.343,Y -670.935,Z 1363.365,A 0.000,B 0.000,C 90.000,E1 101.591} C_DIS
LIN {X 0.005,Y -670.191,Z 1363.361,A 0.000,B 0.000,C 90.000,E1 100.894} C_DIS
LIN {X -0.141,Y -669.525,Z 1363.358,A 0.000,B 0.000,C 90.000,E1 100.423} C_DIS
LIN {X 0.248,Y -668.588,Z 1363.355,A 0.000,B 0.000,C 90.000,E1 99.905} C_DIS
LIN {X -0.022,Y -667.341,Z 1363.353,A 0.000,B 0.000,C 90.000,E1 99.443} C_DIS
LIN {X 0.274,Y -665.062,Z 1363.349,A 0.000,B 0.000,C 90.000,E1 98.690} C_DIS
LIN {X -0.111,Y -662.282,Z 1363.344,A 0.000,B 0.000,C 90.000,E1 97.992} C_DIS
LIN {X 0.243,Y -660.216,Z 1363.342,A 0.000,B 0.000,C 90.000,E1 97.473} C_DIS
LIN {X -0.191,Y -656.835,Z 1363.338,A 0.000,B 0.000,C 90.000,E1 96.777} C_DIS
LIN {X 0.018,Y -653.645,Z 1363.334,A 0.000,B 0.000,C 90.000,E1 96.144} C_DIS
LIN {X 0.152,Y -649.204,Z 1363.330,A 0.000,B 0.000,C 90.000,E1 95.391} C_DIS
LIN {X 0.176,Y -644.480,Z 1363.326,A 0.000,B 0.000,C 90.000,E1 94.645} C_DIS
LIN {X 0.151,Y -639.378,Z 1363.322,A 0.000,B 0.000,C 90.000,E1 93.898} C_DIS
LIN {X 0.293,Y -635.541,Z 1363.319,A 0.000,B 0.000,C 90.000,E1 93.383} C_DIS
LIN {X 0.313,Y -629.901,Z 1363.315,A 0.000,B 0.000,C 90.000,E1 92.751} C_DIS
LIN {X -0.303,Y -623.705,Z 1363.312,A 0.000,B 0.000,C 90.000,E1 92.178} C_DIS
LIN {X -0.229,Y -616.029,Z 1363.308,A 0.000,B 0.000,C 90.000,E1 91.432} C_DIS
LIN {X 0.186,Y -612.031,Z 1363.306,A 0.000,B 0.000,C 90.000,E1 91.031} C_DIS
LIN {X 0.137,Y -609.251,Z 1363.305,A 0.000,B 0.000,C 90.000,E1 90.802} C_DIS
LIN {X 0.280,Y -603.255,Z 1363.302,A 0.000,B 0.000,C 90.000,E1 90.344} C_DIS
LIN {X -0.190,Y -596.476,Z 1363.300,A 0.000,B 0.000,C 90.000,E1 90.000} C_DIS
LIN {X -0.092,Y -589.476,Z 1363.298,A 0.000,B 0.000,C 90.000,E1 89.656} C_DIS
LIN {X -0.168,Y -582.415,Z 1363.297,A 0.000,B 0.000,C 90.000,E1 89.370} C_DIS
LIN {X 0.225,Y -578.489,Z 1363.295,A 0.000,B 0.000,C 90.000,E1 89.141} C_DIS
LIN {X -0.278,Y -576.011,Z 1363.294,A 0.000,B 0.000,C 90.000,E1 89.026} C_DIS
LIN {X -0.270,Y -574.444,Z 1363.294,A 0.000,B 0.000,C 90.000,E1 88.912} C_DIS
LIN {X 0.272,Y -574.403,Z 1363.294,A 0.000,B 0.000,C 90.000,E1 88.854} C_DIS
LIN {X 0.231,Y -573.516,Z 1363.292,A 0.000,B 0.000,C 90.000,E1 88.625} C_DIS
LIN {X 0.158,Y -573.368,Z 1363.290,A 0.000,B 0.000,C 90.000,E1 88.224} C_DIS
LIN {X 0.195,Y -575.888,Z 1363.274,A 0.000,B 0.000,C 90.000,E1 85.241} C_DIS
LIN {X 0.055,Y -577.664,Z 1363.265,A 0.000,B 0.000,C 90.000,E1 83.628} C_DIS
LIN {X 0.163,Y -579.921,Z 1363.254,A 0.000,B 0.000,C 90.000,E1 81.724} C_DIS
LIN {X 0.044,Y -581.548,Z 1363.247,A 0.000,B 0.000,C 90.000,E1 80.387} C_DIS
LIN {X -0.046,Y -583.027,Z 1363.239,A 0.000,B 0.000,C 90.000,E1 79.050} C_DIS
LIN {X -0.239,Y -584.085,Z 1363.233,A 0.000,B 0.000,C 90.000,E1 77.993} C_DIS
LIN {X 0.071,Y -585.603,Z 1363.224,A 0.000,B 0.000,C 90.000,E1 76.353} C_DIS
LIN {X -0.025,Y -586.788,Z 1363.215,A 0.000,B 0.000,C 90.000,E1 74.755} C_DIS
LIN {X -0.025,Y -587.477,Z 1363.209,A 0.000,B 0.000,C 90.000,E1 73.685} C_DIS
LIN {X 0.252,Y -588.512,Z 1363.200,A 0.000,B 0.000,C 90.000,E1 72.054} C_DIS
LIN {X 0.232,Y -589.561,Z 1363.190,A 0.000,B 0.000,C 90.000,E1 70.188} C_DIS
LIN {X 0.083,Y -590.669,Z 1363.180,A 0.000,B 0.000,C 90.000,E1 68.337} C_DIS
LIN {X -0.139,Y -592.171,Z 1363.168,A 0.000,B 0.000,C 90.000,E1 66.230} C_DIS
LIN {X 0.096,Y -593.514,Z 1363.159,A 0.000,B 0.000,C 90.000,E1 64.613} C_DIS
LIN {X 0.328,Y -594.698,Z 1363.150,A 0.000,B 0.000,C 90.000,E1 62.999} C_DIS
LIN {X -0.018,Y -596.167,Z 1363.140,A 0.000,B 0.000,C 90.000,E1 61.179} C_DIS
LIN {X 0.051,Y -597.634,Z 1363.131,A 0.000,B 0.000,C 90.000,E1 59.587} C_DIS
LIN {X -0.079,Y -598.919,Z 1363.124,A 0.000,B 0.000,C 90.000,E1 58.280} C_DIS
LIN {X -0.068,Y -600.198,Z 1363.116,A 0.000,B 0.000,C 90.000,E1 56.962} C_DIS
LIN {X 0.231,Y -601.183,Z 1363.111,A 0.000,B 0.000,C 90.000,E1 55.881} C_DIS
LIN {X -0.052,Y -602.848,Z 1363.100,A 0.000,B 0.000,C 90.000,E1 54.069} C_DIS
LIN {X 0.123,Y -603.848,Z 1363.095,A 0.000,B 0.000,C 90.000,E1 53.004} C_DIS
LIN {X -0.169,Y -604.716,Z 1363.089,A 0.000,B 0.000,C 90.000,E1 51.984} C_DIS
LIN {X 0.195,Y -605.575,Z 1363.082,A 0.000,B 0.000,C 90.000,E1 50.642} C_DIS
LIN {X -0.016,Y -606.430,Z 1363.073,A 0.000,B 0.000,C 90.000,E1 49.094} C_DIS
LIN {X 0.108,Y -606.804,Z 1363.067,A 0.000,B 0.000,C 90.000,E1 48.038} C_DIS
LIN {X 0.009,Y -607.100,Z 1363.060,A 0.000,B 0.000,C 90.000,E1 46.743} C_DIS
LIN {X -0.061,Y -607.210,Z 1363.052,A 0.000,B 0.000,C 90.000,E1 45.445} C_DIS
LIN {X 0.285,Y -607.047,Z 1363.045,A 0.000,B 0.000,C 90.000,E1 44.109} C_DIS
LIN {X -0.031,Y -606.663,Z 1363.039,A 0.000,B 0.000,C 90.000,E1 43.095} C_DIS
LIN {X 0.117,Y -605.935,Z 1363.031,A 0.000,B 0.000,C 90.000,E1 41.515} C_DIS
LIN {X -0.024,Y -605.564,Z 1363.026,A 0.000,B 0.000,C 90.000,E1 40.744} C_DIS
LIN {X -0.040,Y -604.732,Z 1363.019,A 0.000,B 0.000,C 90.000,E1 39.439} C_DIS
LIN {X 0.321,Y -603.771,Z 1363.012,A 0.000,B 0.000,C 90.000,E1 38.096} C_DIS
LIN {X -0.230,Y -603.083,Z 1363.007,A 0.000,B 0.000,C 90.000,E1 37.363} C_DIS
LIN {X -0.054,Y -601.940,Z 1363.002,A 0.000,B 0.000,C 90.000,E1 36.297} C_DIS
LIN {X 0.006,Y -599.867,Z 1362.994,A 0.000,B 0.000,C 90.000,E1 34.978} C_DIS
LIN {X 0.134,Y -597.670,Z 1362.989,A 0.000,B 0.000,C 90.000,E1 33.913} C_DIS
LIN {X -0.333,Y -595.898,Z 1362.984,A 0.000,B 0.000,C 90.000,E1 33.166} C_DIS
LIN {X 0.006,Y -594.001,Z 1362.980,A 0.000,B 0.000,C 90.000,E1 32.339} C_DIS
LIN {X 0.009,Y -591.697,Z 1362.975,A 0.000,B 0.000,C 90.000,E1 31.544} C_DIS
LIN {X -0.008,Y -589.104,Z 1362.971,A 0.000,B 0.000,C 90.000,E1 30.747} C_DIS
LIN {X 0.068,Y -587.172,Z 1362.968,A 0.000,B 0.000,C 90.000,E1 30.207} C_DIS
LIN {X 0.004,Y -584.075,Z 1362.964,A 0.000,B 0.000,C 90.000,E1 29.411} C_DIS
LIN {X 0.037,Y -581.835,Z 1362.960,A 0.000,B 0.000,C 90.000,E1 28.871} C_DIS
LIN {X -0.297,Y -578.631,Z 1362.957,A 0.000,B 0.000,C 90.000,E1 28.231} C_DIS
LIN {X 0.124,Y -575.291,Z 1362.953,A 0.000,B 0.000,C 90.000,E1 27.513} C_DIS
LIN {X 0.169,Y -570.903,Z 1362.948,A 0.000,B 0.000,C 90.000,E1 26.693} C_DIS
LIN {X -0.079,Y -568.567,Z 1362.946,A 0.000,B 0.000,C 90.000,E1 26.309} C_DIS
LIN {X 0.329,Y -565.244,Z 1362.943,A 0.000,B 0.000,C 90.000,E1 25.720} C_DIS
LIN {X 0.270,Y -559.951,Z 1362.938,A 0.000,B 0.000,C 90.000,E1 24.899} C_DIS
LIN {X 0.263,Y -555.089,Z 1362.935,A 0.000,B 0.000,C 90.000,E1 24.207} C_DIS
LIN {X -0.025,Y -547.641,Z 1362.929,A 0.000,B 0.000,C 90.000,E1 23.259} C_DIS
LIN {X -0.110,Y -539.478,Z 1362.924,A 0.000,B 0.000,C 90.000,E1 22.280} C_DIS
LIN {X 0.196,Y -533.315,Z 1362.920,A 0.000,B 0.000,C 90.000,E1 21.535} C_DIS
LIN {X 0.118,Y -523.007,Z 1362.914,A 0.000,B 0.000,C 90.000,E1 20.429} C_DIS
LIN {X 0.110,Y -512.417,Z 1362.907,A 0.000,B 0.000,C 90.000,E1 19.322} C_DIS
LIN {X -0.071,Y -501.753,Z 1362.901,A 0.000,B 0.000,C 90.000,E1 18.236} C_DIS
LIN {X -0.183,Y -493.592,Z 1362.897,A 0.000,B 0.000,C 90.000,E1 17.402} C_DIS
LIN {X -0.165,Y -482.350,Z 1362.891,A 0.000,B 0.000,C 90.000,E1 16.315} C_DIS
LIN {X -0.131,Y -466.757,Z 1362.882,A 0.000,B 0.000,C 90.000,E1 14.773} C_DIS
LIN {X 0.085,Y -454.001,Z 1362.875,A 0.000,B 0.000,C 90.000,E1 13.480} C_DIS
LIN {X 0.161,Y -436.976,Z 1362.865,A 0.000,B 0.000,C 90.000,E1 11.715} C_DIS
LIN {X -0.014,Y -420.430,Z 1362.855,A 0.000,B 0.000,C 90.000,E1 9.905} C_DIS
LIN {X -0.171,Y -406.537,Z 1362.846,A 0.000,B 0.000,C 90.000,E1 8.333} C_DIS
LIN {X -0.196,Y -396.661,Z 1362.840,A 0.000,B 0.000,C 90.000,E1 7.182} C_DIS
LIN {X 0.026,Y -393.058,Z 1362.837,A 0.000,B 0.000,C 90.000,E1 6.606} C_DIS
LIN {X -0.011,Y -393.029,Z 1362.837,A 0.000,B 0.000,C 90.000,E1 6.606} C_DIS
LIN {X -0.125,Y -394.108,Z 1362.836,A 0.000,B 0.000,C 90.000,E1 6.429} C_DIS
LIN {X 0.049,Y -394.759,Z 1362.835,A 0.000,B 0.000,C 90.000,E1 6.315} C_DIS
LIN {X -0.078,Y -398.918,Z 1362.833,A 0.000,B 0.000,C 90.000,E1 5.967} C_DIS
LIN {X -0.049,Y -410.954,Z 1362.828,A 0.000,B 0.000,C 90.000,E1 5.106} C_DIS
LIN {X 0.047,Y -417.106,Z 1362.826,A 0.000,B 0.000,C 90.000,E1 4.588} C_DIS
LIN {X -0.181,Y -422.972,Z 1362.823,A 0.000,B 0.000,C 90.000,E1 4.069} C_DIS
LIN {X -0.217,Y -429.891,Z 1362.818,A 0.000,B 0.000,C 90.000,E1 3.326} C_DIS
LIN {X -0.190,Y -436.648,Z 1362.814,A 0.000,B 0.000,C 90.000,E1 2.522} C_DIS
LIN {X 0.088,Y -442.800,Z 1362.810,A 0.000,B 0.000,C 90.000,E1 1.718} C_DIS
LIN {X -0.034,Y -449.008,Z 1362.805,A 0.000,B 0.000,C 90.000,E1 0.917} C_DIS
LIN {X -0.096,Y -454.810,Z 1362.801,A 0.000,B 0.000,C 90.000,E1 0.115} C_DIS
LIN {X 0.091,Y -461.127,Z 1362.795,A 0.000,B 0.000,C 90.000,E1 359.141} C_DIS
LIN {X 0.040,Y -465.168,Z 1362.792,A 0.000,B 0.000,C 90.000,E1 358.511} C_DIS
LIN {X -0.201,Y -470.690,Z 1362.786,A 0.000,B 0.000,C 90.000,E1 357.593} C_DIS
LIN {X -0.185,Y -474.110,Z 1362.783,A 0.000,B 0.000,C 90.000,E1 356.963} C_DIS
LIN {X 0.016,Y -478.119,Z 1362.779,A 0.000,B 0.000,C 90.000,E1 356.159} C_DIS
LIN {X -0.223,Y -481.745,Z 1362.774,A 0.000,B 0.000,C 90.000,E1 355.412} C_DIS
LIN {X -0.093,Y -484.471,Z 1362.771,A 0.000,B 0.000,C 90.000,E1 354.780} C_DIS
LIN {X 0.060,Y -487.023,Z 1362.768,A 0.000,B 0.000,C 90.000,E1 354.147} C_DIS
LIN {X 0.104,Y -490.428,Z 1362.762,A 0.000,B 0.000,C 90.000,E1 353.223} C_DIS
LIN {X -0.190,Y -492.559,Z 1362.759,A 0.000,B 0.000,C 90.000,E1 352.648} C_DIS
LIN {X 0.084,Y -494.482,Z 1362.756,A 0.000,B 0.000,C 90.000,E1 352.008} C_DIS
LIN {X 0.213,Y -497.074,Z 1362.751,A 0.000,B 0.000,C 90.000,E1 351.084} C_DIS
LIN {X -0.208,Y -500.183,Z 1362.744,A 0.000,B 0.000,C 90.000,E1 349.926} C_DIS
LIN {X 0.060,Y -502.235,Z 1362.739,A 0.000,B 0.000,C 90.000,E1 348.993} C_DIS
LIN {X -0.097,Y -504.619,Z 1362.732,A 0.000,B 0.000,C 90.000,E1 347.813} C_DIS
LIN {X 0.225,Y -506.161,Z 1362.727,A 0.000,B 0.000,C 90.000,E1 346.881} C_DIS
LIN {X 0.134,Y -508.035,Z 1362.721,A 0.000,B 0.000,C 90.000,E1 345.700} C_DIS
LIN {X 0.066,Y -509.387,Z 1362.714,A 0.000,B 0.000,C 90.000,E1 344.519} C_DIS
LIN {X 0.155,Y -509.617,Z 1362.712,A 0.000,B 0.000,C 90.000,E1 344.212} C_DIS
LIN {X 0.107,Y -509.673,Z 1362.711,A 0.000,B 0.000,C 90.000,E1 343.921} C_DIS
LIN {X 0.202,Y -509.576,Z 1362.709,A 0.000,B 0.000,C 90.000,E1 343.614} C_DIS
LIN {X 0.153,Y -509.188,Z 1362.708,A 0.000,B 0.000,C 90.000,E1 343.323} C_DIS
LIN {X 0.100,Y -508.403,Z 1362.706,A 0.000,B 0.000,C 90.000,E1 343.032} C_DIS
LIN {X -0.095,Y -507.707,Z 1362.705,A 0.000,B 0.000,C 90.000,E1 342.906} C_DIS
LIN {X 0.194,Y -506.373,Z 1362.704,A 0.000,B 0.000,C 90.000,E1 342.725} C_DIS
LIN {X 0.112,Y -474.093,Z 1362.698,A 0.000,B 0.000,C 90.000,E1 341.529} C_DIS
LIN {X -0.105,Y -443.184,Z 1362.690,A 0.000,B 0.000,C 90.000,E1 340.242} C_DIS
LIN {X 0.006,Y -415.961,Z 1362.683,A 0.000,B 0.000,C 90.000,E1 338.901} C_DIS
LIN {X 0.025,Y -390.600,Z 1362.675,A 0.000,B 0.000,C 90.000,E1 337.486} C_DIS
LIN {X 0.081,Y -368.857,Z 1362.667,A 0.000,B 0.000,C 90.000,E1 336.102} C_DIS
LIN {X -0.158,Y -363.038,Z 1362.665,A 0.000,B 0.000,C 90.000,E1 335.741} C_DIS
LIN {X -0.031,Y -362.993,Z 1362.665,A 0.000,B 0.000,C 90.000,E1 335.717} C_DIS
LIN {X -0.026,Y -366.089,Z 1362.642,A 0.000,B 0.000,C 90.000,E1 331.563} C_DIS
LIN {X 0.018,Y -370.648,Z 1362.607,A 0.000,B 0.000,C 90.000,E1 325.261} C_DIS
LIN {X 0.063,Y -371.828,Z 1362.601,A 0.000,B 0.000,C 90.000,E1 324.149} C_DIS
LIN {X 0.080,Y -377.498,Z 1362.566,A 0.000,B 0.000,C 90.000,E1 317.919} C_DIS
LIN {X 0.092,Y -377.977,Z 1362.564,A 0.000,B 0.000,C 90.000,E1 317.553} C_DIS
LIN {X 0.114,Y -378.803,Z 1362.558,A 0.000,B 0.000,C 90.000,E1 316.458} C_DIS
LIN {X -0.137,Y -384.585,Z 1362.528,A 0.000,B 0.000,C 90.000,E1 311.067} C_DIS
LIN {X -0.093,Y -384.963,Z 1362.526,A 0.000,B 0.000,C 90.000,E1 310.701} C_DIS
LIN {X 0.078,Y -390.757,Z 1362.494,A 0.000,B 0.000,C 90.000,E1 304.945} C_DIS
LIN {X -0.078,Y -391.249,Z 1362.492,A 0.000,B 0.000,C 90.000,E1 304.612} C_DIS
LIN {X 0.076,Y -396.963,Z 1362.459,A 0.000,B 0.000,C 90.000,E1 298.565} C_DIS
LIN {X 0.027,Y -401.327,Z 1362.428,A 0.000,B 0.000,C 90.000,E1 292.950} C_DIS
LIN {X 0.108,Y -401.654,Z 1362.426,A 0.000,B 0.000,C 90.000,E1 292.589} C_DIS
LIN {X -0.127,Y -404.739,Z 1362.395,A 0.000,B 0.000,C 90.000,E1 287.040} C_DIS
LIN {X -0.124,Y -406.152,Z 1362.364,A 0.000,B 0.000,C 90.000,E1 281.478} C_DIS
LIN {X -0.026,Y -405.683,Z 1362.333,A 0.000,B 0.000,C 90.000,E1 275.910} C_DIS
LIN {X 0.046,Y -403.568,Z 1362.306,A 0.000,B 0.000,C 90.000,E1 271.031} C_DIS
LIN {X -0.019,Y -403.196,Z 1362.302,A 0.000,B 0.000,C 90.000,E1 270.344} C_DIS
LIN {X -0.185,Y -399.073,Z 1362.273,A 0.000,B 0.000,C 90.000,E1 265.122} C_DIS
LIN {X 0.155,Y -398.795,Z 1362.271,A 0.000,B 0.000,C 90.000,E1 264.723} C_DIS
LIN {X 0.045,Y -393.303,Z 1362.243,A 0.000,B 0.000,C 90.000,E1 259.803} C_DIS
LIN {X -0.035,Y -392.694,Z 1362.240,A 0.000,B 0.000,C 90.000,E1 259.106} C_DIS
LIN {X 0.135,Y -386.262,Z 1362.214,A 0.000,B 0.000,C 90.000,E1 254.448} C_DIS
LIN {X 0.100,Y -385.164,Z 1362.208,A 0.000,B 0.000,C 90.000,E1 253.378} C_DIS
LIN {X -0.016,Y -377.379,Z 1362.180,A 0.000,B 0.000,C 90.000,E1 248.337} C_DIS
LIN {X 0.080,Y -376.105,Z 1362.174,A 0.000,B 0.000,C 90.000,E1 247.230} C_DIS
LIN {X -0.192,Y -368.772,Z 1362.149,A 0.000,B 0.000,C 90.000,E1 242.871} C_DIS
LIN {X -0.057,Y -366.415,Z 1362.139,A 0.000,B 0.000,C 90.000,E1 241.001} C_DIS
LIN {X -0.032,Y -365.129,Z 1362.135,A 0.000,B 0.000,C 90.000,E1 240.255} C_DIS
LIN {X 0.034,Y -358.523,Z 1362.112,A 0.000,B 0.000,C 90.000,E1 236.135} C_DIS
LIN {X -0.114,Y -356.195,Z 1362.101,A 0.000,B 0.000,C 90.000,E1 234.276} C_DIS
LIN {X 0.033,Y -354.958,Z 1362.097,A 0.000,B 0.000,C 90.000,E1 233.497} C_DIS
LIN {X 0.016,Y -348.178,Z 1362.072,A 0.000,B 0.000,C 90.000,E1 228.933} C_DIS
LIN {X -0.050,Y -346.071,Z 1362.061,A 0.000,B 0.000,C 90.000,E1 227.025} C_DIS
LIN {X 0.066,Y -339.697,Z 1362.036,A 0.000,B 0.000,C 90.000,E1 222.366} C_DIS
LIN {X -0.120,Y -336.690,Z 1362.018,A 0.000,B 0.000,C 90.000,E1 219.277} C_DIS
LIN {X -0.209,Y -330.770,Z 1361.988,A 0.000,B 0.000,C 90.000,E1 213.785} C_DIS
LIN {X -0.080,Y -329.215,Z 1361.974,A 0.000,B 0.000,C 90.000,E1 211.386} C_DIS
LIN {X -0.070,Y -325.894,Z 1361.953,A 0.000,B 0.000,C 90.000,E1 207.641} C_DIS
LIN {X -0.088,Y -325.928,Z 1361.953,A 0.000,B 0.000,C 90.000,E1 207.641} C_DIS
LIN {X 0.174,Y -345.315,Z 1361.945,A 0.000,B 0.000,C 90.000,E1 205.976} C_DIS
LIN {X -0.063,Y -365.629,Z 1361.936,A 0.000,B 0.000,C 90.000,E1 204.515} C_DIS
LIN {X -0.151,Y -387.870,Z 1361.928,A 0.000,B 0.000,C 90.000,E1 203.078} C_DIS
LIN {X 0.028,Y -412.068,Z 1361.920,A 0.000,B 0.000,C 90.000,E1 201.663} C_DIS
LIN {X -0.066,Y -438.228,Z 1361.913,A 0.000,B 0.000,C 90.000,E1 200.355} C_DIS
LIN {X 0.211,Y -445.236,Z 1361.911,A 0.000,B 0.000,C 90.000,E1 199.993} C_DIS
LIN {X -0.039,Y -447.872,Z 1361.910,A 0.000,B 0.000,C 90.000,E1 199.866} C_DIS
LIN {X 0.220,Y -449.211,Z 1361.909,A 0.000,B 0.000,C 90.000,E1 199.631} C_DIS
LIN {X 0.092,Y -450.491,Z 1361.907,A 0.000,B 0.000,C 90.000,E1 199.322} C_DIS
LIN {X -0.178,Y -451.369,Z 1361.906,A 0.000,B 0.000,C 90.000,E1 199.033} C_DIS
LIN {X 0.131,Y -452.018,Z 1361.904,A 0.000,B 0.000,C 90.000,E1 198.671} C_DIS
LIN {X -0.102,Y -452.784,Z 1361.900,A 0.000,B 0.000,C 90.000,E1 198.055} C_DIS
LIN {X -0.154,Y -453.663,Z 1361.895,A 0.000,B 0.000,C 90.000,E1 197.094} C_DIS
LIN {X 0.085,Y -455.097,Z 1361.884,A 0.000,B 0.000,C 90.000,E1 195.134} C_DIS
LIN {X 0.035,Y -456.210,Z 1361.875,A 0.000,B 0.000,C 90.000,E1 193.536} C_DIS
LIN {X -0.100,Y -457.292,Z 1361.866,A 0.000,B 0.000,C 90.000,E1 191.951} C_DIS
LIN {X 0.228,Y -458.280,Z 1361.858,A 0.000,B 0.000,C 90.000,E1 190.310} C_DIS
LIN {X 0.018,Y -458.790,Z 1361.852,A 0.000,B 0.000,C 90.000,E1 189.378} C_DIS
LIN {X 0.210,Y -459.425,Z 1361.843,A 0.000,B 0.000,C 90.000,E1 187.757} C_DIS
LIN {X 0.177,Y -459.843,Z 1361.836,A 0.000,B 0.000,C 90.000,E1 186.486} C_DIS
LIN {X 0.099,Y -460.099,Z 1361.829,A 0.000,B 0.000,C 90.000,E1 185.220} C_DIS
LIN {X 0.023,Y -460.029,Z 1361.822,A 0.000,B 0.000,C 90.000,E1 183.955} C_DIS
LIN {X -0.084,Y -459.921,Z 1361.815,A 0.000,B 0.000,C 90.000,E1 182.694} C_DIS
LIN {X -0.194,Y -459.452,Z 1361.808,A 0.000,B 0.000,C 90.000,E1 181.432} C_DIS
LIN {X -0.059,Y -458.870,Z 1361.803,A 0.000,B 0.000,C 90.000,E1 180.458} C_DIS
LIN {X 0.071,Y -457.856,Z 1361.797,A 0.000,B 0.000,C 90.000,E1 179.484} C_DIS
LIN {X -0.085,Y -456.005,Z 1361.790,A 0.000,B 0.000,C 90.000,E1 178.224} C_DIS
LIN {X 0.020,Y -453.988,Z 1361.785,A 0.000,B 0.000,C 90.000,E1 177.249} C_DIS
LIN {X 0.103,Y -451.405,Z 1361.779,A 0.000,B 0.000,C 90.000,E1 176.274} C_DIS
LIN {X 0.004,Y -449.473,Z 1361.776,A 0.000,B 0.000,C 90.000,E1 175.641} C_DIS
LIN {X 0.027,Y -445.710,Z 1361.770,A 0.000,B 0.000,C 90.000,E1 174.666} C_DIS
LIN {X -0.180,Y -443.570,Z 1361.768,A 0.000,B 0.000,C 90.000,E1 174.204} C_DIS
LIN {X 0.043,Y -441.146,Z 1361.765,A 0.000,B 0.000,C 90.000,E1 173.685} C_DIS
LIN {X -0.137,Y -437.680,Z 1361.761,A 0.000,B 0.000,C 90.000,E1 173.053} C_DIS
LIN {X 0.178,Y -432.744,Z 1361.757,A 0.000,B 0.000,C 90.000,E1 172.186} C_DIS
LIN {X 0.098,Y -426.070,Z 1361.751,A 0.000,B 0.000,C 90.000,E1 171.197} C_DIS
LIN {X 0.077,Y -414.385,Z 1361.742,A 0.000,B 0.000,C 90.000,E1 169.511} C_DIS
LIN {X -0.184,Y -405.487,Z 1361.734,A 0.000,B 0.000,C 90.000,E1 168.173} C_DIS
LIN {X -0.020,Y -396.964,Z 1361.726,A 0.000,B 0.000,C 90.000,E1 166.756} C_DIS
LIN {X -0.082,Y -393.458,Z 1361.723,A 0.000,B 0.000,C 90.000,E1 166.061} C_DIS
LIN {X -0.055,Y -392.797,Z 1361.722,A 0.000,B 0.000,C 90.000,E1 165.880} C_DIS
LIN {X 0.110,Y -391.310,Z 1361.718,A 0.000,B 0.000,C 90.000,E1 165.283} C_DIS
LIN {X -0.134,Y -391.122,Z 1361.717,A 0.000,B 0.000,C 90.000,E1 164.991} C_DIS
LIN {X -0.172,Y -391.132,Z 1361.717,A 0.000,B 0.000,C 90.000,E1 164.991} C_DIS
LIN {X 0.075,Y -392.466,Z 1361.715,A 0.000,B 0.000,C 90.000,E1 164.755} C_DIS
LIN {X -0.134,Y -393.888,Z 1361.714,A 0.000,B 0.000,C 90.000,E1 164.519} C_DIS
LIN {X -0.181,Y -398.786,Z 1361.711,A 0.000,B 0.000,C 90.000,E1 163.921} C_DIS
LIN {X 0.118,Y -404.025,Z 1361.708,A 0.000,B 0.000,C 90.000,E1 163.323} C_DIS
LIN {X 0.132,Y -413.036,Z 1361.703,A 0.000,B 0.000,C 90.000,E1 162.489} C_DIS
LIN {X 0.151,Y -433.585,Z 1361.693,A 0.000,B 0.000,C 90.000,E1 160.786} C_DIS
LIN {X 0.100,Y -452.705,Z 1361.685,A 0.000,B 0.000,C 90.000,E1 159.337} C_DIS
LIN {X -0.211,Y -458.942,Z 1361.683,A 0.000,B 0.000,C 90.000,E1 158.901} C_DIS
LIN {X -0.136,Y -466.507,Z 1361.679,A 0.000,B 0.000,C 90.000,E1 158.284} C_DIS
LIN {X -0.231,Y -474.007,Z 1361.676,A 0.000,B 0.000,C 90.000,E1 157.667} C_DIS
LIN {X 0.160,Y -481.374,Z 1361.672,A 0.000,B 0.000,C 90.000,E1 156.975} C_DIS
LIN {X 0.173,Y -489.936,Z 1361.668,A 0.000,B 0.000,C 90.000,E1 156.177} C_DIS
LIN {X -0.053,Y -495.514,Z 1361.665,A 0.000,B 0.000,C 90.000,E1 155.665} C_DIS
LIN {X -0.135,Y -503.754,Z 1361.660,A 0.000,B 0.000,C 90.000,E1 154.845} C_DIS
LIN {X 0.135,Y -510.137,Z 1361.656,A 0.000,B 0.000,C 90.000,E1 154.101} C_DIS
LIN {X -0.207,Y -517.593,Z 1361.651,A 0.000,B 0.000,C 90.000,E1 153.256} C_DIS
LIN {X 0.118,Y -523.123,Z 1361.647,A 0.000,B 0.000,C 90.000,E1 152.487} C_DIS
LIN {X -0.118,Y -526.240,Z 1361.645,A 0.000,B 0.000,C 90.000,E1 152.076} C_DIS
LIN {X -0.272,Y -529.981,Z 1361.642,A 0.000,B 0.000,C 90.000,E1 151.513} C_DIS
LIN {X -0.300,Y -533.760,Z 1361.638,A 0.000,B 0.000,C 90.000,E1 150.795} C_DIS
LIN {X -0.150,Y -536.414,Z 1361.634,A 0.000,B 0.000,C 90.000,E1 150.205} C_DIS
LIN {X 0.016,Y -538.743,Z 1361.631,A 0.000,B 0.000,C 90.000,E1 149.616} C_DIS
LIN {X -0.266,Y -540.745,Z 1361.628,A 0.000,B 0.000,C 90.000,E1 149.076} C_DIS
LIN {X -0.058,Y -543.494,Z 1361.623,A 0.000,B 0.000,C 90.000,E1 148.201} C_DIS
LIN {X 0.180,Y -545.624,Z 1361.619,A 0.000,B 0.000,C 90.000,E1 147.327} C_DIS
LIN {X -0.054,Y -546.824,Z 1361.615,A 0.000,B 0.000,C 90.000,E1 146.786} C_DIS
LIN {X -0.196,Y -548.827,Z 1361.609,A 0.000,B 0.000,C 90.000,E1 145.674} C_DIS
LIN {X -0.099,Y -549.690,Z 1361.606,A 0.000,B 0.000,C 90.000,E1 145.102} C_DIS
LIN {X -0.198,Y -551.109,Z 1361.600,A 0.000,B 0.000,C 90.000,E1 143.989} C_DIS
LIN {X -0.019,Y -551.962,Z 1361.595,A 0.000,B 0.000,C 90.000,E1 143.130} C_DIS
LIN {X -0.068,Y -553.268,Z 1361.586,A 0.000,B 0.000,C 90.000,E1 141.457} C_DIS
LIN {X 0.258,Y -554.334,Z 1361.577,A 0.000,B 0.000,C 90.000,E1 139.747} C_DIS
LIN {X -0.250,Y -555.194,Z 1361.569,A 0.000,B 0.000,C 90.000,E1 138.405} C_DIS
LIN {X -0.007,Y -555.852,Z 1361.561,A 0.000,B 0.000,C 90.000,E1 136.986} C_DIS
LIN {X 0.253,Y -556.484,Z 1361.553,A 0.000,B 0.000,C 90.000,E1 135.567} C_DIS
LIN {X -0.217,Y -557.196,Z 1361.544,A 0.000,B 0.000,C 90.000,E1 133.947} C_DIS
LIN {X 0.137,Y -558.183,Z 1361.535,A 0.000,B 0.000,C 90.000,E1 132.243} C_DIS
LIN {X 0.022,Y -558.664,Z 1361.532,A 0.000,B 0.000,C 90.000,E1 131.838} C_DIS
LIN {X -0.095,Y -559.538,Z 1361.530,A 0.000,B 0.000,C 90.000,E1 131.434} C_DIS
LIN {X -0.014,Y -560.011,Z 1361.529,A 0.000,B 0.000,C 90.000,E1 131.148} C_DIS
LIN {X -0.358,Y -560.143,Z 1361.528,A 0.000,B 0.000,C 90.000,E1 131.148} C_DIS
LIN {X 0.021,Y -560.168,Z 1361.528,A 0.000,B 0.000,C 90.000,E1 131.105} C_DIS
LIN {X 0.189,Y -561.701,Z 1361.528,A 0.000,B 0.000,C 90.000,E1 130.987} C_DIS
LIN {X 0.115,Y -562.928,Z 1361.528,A 0.000,B 0.000,C 90.000,E1 130.943} C_DIS
LIN {X 0.106,Y -578.261,Z 1361.525,A 0.000,B 0.000,C 90.000,E1 130.458} C_DIS
LIN {X -0.102,Y -584.347,Z 1361.523,A 0.000,B 0.000,C 90.000,E1 130.216} C_DIS
LIN {X 0.041,Y -590.003,Z 1361.522,A 0.000,B 0.000,C 90.000,E1 129.886} C_DIS
LIN {X 0.221,Y -595.705,Z 1361.520,A 0.000,B 0.000,C 90.000,E1 129.483} C_DIS
LIN {X -0.110,Y -600.005,Z 1361.518,A 0.000,B 0.000,C 90.000,E1 129.197} C_DIS
LIN {X -0.068,Y -605.466,Z 1361.515,A 0.000,B 0.000,C 90.000,E1 128.749} C_DIS
LIN {X 0.165,Y -610.650,Z 1361.513,A 0.000,B 0.000,C 90.000,E1 128.257} C_DIS
LIN {X 0.147,Y -616.957,Z 1361.509,A 0.000,B 0.000,C 90.000,E1 127.649} C_DIS
LIN {X -0.010,Y -623.040,Z 1361.506,A 0.000,B 0.000,C 90.000,E1 127.030} C_DIS
LIN {X 0.145,Y -628.805,Z 1361.502,A 0.000,B 0.000,C 90.000,E1 126.377} C_DIS
LIN {X 0.349,Y -634.303,Z 1361.499,A 0.000,B 0.000,C 90.000,E1 125.724} C_DIS
LIN {X 0.226,Y -639.476,Z 1361.495,A 0.000,B 0.000,C 90.000,E1 125.105} C_DIS
LIN {X -0.359,Y -645.129,Z 1361.491,A 0.000,B 0.000,C 90.000,E1 124.405} C_DIS
LIN {X 0.002,Y -650.424,Z 1361.487,A 0.000,B 0.000,C 90.000,E1 123.627} C_DIS
LIN {X -0.390,Y -653.686,Z 1361.484,A 0.000,B 0.000,C 90.000,E1 123.166} C_DIS
LIN {X -0.354,Y -657.372,Z 1361.481,A 0.000,B 0.000,C 90.000,E1 122.546} C_DIS
LIN {X 0.269,Y -660.646,Z 1361.477,A 0.000,B 0.000,C 90.000,E1 121.878} C_DIS
LIN {X -0.051,Y -662.963,Z 1361.475,A 0.000,B 0.000,C 90.000,E1 121.416} C_DIS
LIN {X 0.123,Y -666.056,Z 1361.470,A 0.000,B 0.000,C 90.000,E1 120.669} C_DIS
LIN {X -0.014,Y -668.502,Z 1361.466,A 0.000,B 0.000,C 90.000,E1 119.951} C_DIS
LIN {X -0.218,Y -671.186,Z 1361.461,A 0.000,B 0.000,C 90.000,E1 118.999} C_DIS
LIN {X 0.283,Y -672.302,Z 1361.457,A 0.000,B 0.000,C 90.000,E1 118.231} C_DIS
LIN {X 0.208,Y -672.693,Z 1361.453,A 0.000,B 0.000,C 90.000,E1 117.513} C_DIS
LIN {X 0.131,Y -672.625,Z 1361.449,A 0.000,B 0.000,C 90.000,E1 116.796} C_DIS
LIN {X -0.074,Y -672.210,Z 1361.444,A 0.000,B 0.000,C 90.000,E1 115.848} C_DIS
LIN {X 0.157,Y -671.495,Z 1361.440,A 0.000,B 0.000,C 90.000,E1 115.103} C_DIS
LIN {X -0.110,Y -670.781,Z 1361.437,A 0.000,B 0.000,C 90.000,E1 114.643} C_DIS
LIN {X -0.052,Y -669.308,Z 1361.434,A 0.000,B 0.000,C 90.000,E1 114.155} C_DIS
LIN {X 0.111,Y -668.183,Z 1361.433,A 0.000,B 0.000,C 90.000,E1 113.898} C_DIS
LIN {X -0.189,Y -664.990,Z 1361.430,A 0.000,B 0.000,C 90.000,E1 113.439} C_DIS
LIN {X -0.379,Y -663.744,Z 1361.429,A 0.000,B 0.000,C 90.000,E1 113.334} C_DIS
LIN {X 0.250,Y -659.332,Z 1361.428,A 0.000,B 0.000,C 90.000,E1 112.950} C_DIS
LIN {X 0.289,Y -656.660,Z 1361.427,A 0.000,B 0.000,C 90.000,E1 112.770} C_DIS
LIN {X 0.128,Y -651.707,Z 1361.426,A 0.000,B 0.000,C 90.000,E1 112.589} C_DIS
LIN {X 0.072,Y -647.719,Z 1361.425,A 0.000,B 0.000,C 90.000,E1 112.461} C_DIS
LIN {X -0.157,Y -642.242,Z 1361.424,A 0.000,B 0.000,C 90.000,E1 112.333} C_DIS
LIN {X -0.158,Y -631.638,Z 1361.423,A 0.000,B 0.000,C 90.000,E1 112.078} C_DIS
LIN {X -0.217,Y -631.527,Z 1361.423,A 0.000,B 0.000,C 90.000,E1 112.078} C_DIS
LIN {X 0.187,Y -631.963,Z 1361.422,A 0.000,B 0.000,C 90.000,E1 111.972} C_DIS
LIN {X -0.345,Y -640.257,Z 1361.417,A 0.000,B 0.000,C 90.000,E1 111.046} C_DIS
LIN {X -0.285,Y -644.337,Z 1361.414,A 0.000,B 0.000,C 90.000,E1 110.556} C_DIS
LIN {X -0.168,Y -647.830,Z 1361.411,A 0.000,B 0.000,C 90.000,E1 110.047} C_DIS
LIN {X 0.141,Y -650.835,Z 1361.409,A 0.000,B 0.000,C 90.000,E1 109.523} C_DIS
LIN {X 0.121,Y -654.143,Z 1361.405,A 0.000,B 0.000,C 90.000,E1 108.906} C_DIS
LIN {X -0.004,Y -658.152,Z 1361.400,A 0.000,B 0.000,C 90.000,E1 108.055} C_DIS
LIN {X -0.243,Y -662.282,Z 1361.395,A 0.000,B 0.000,C 90.000,E1 107.094} C_DIS
LIN {X 0.294,Y -665.047,Z 1361.391,A 0.000,B 0.000,C 90.000,E1 106.315} C_DIS
LIN {X 0.037,Y -667.423,Z 1361.387,A 0.000,B 0.000,C 90.000,E1 105.607} C_DIS
LIN {X -0.118,Y -668.676,Z 1361.384,A 0.000,B 0.000,C 90.000,E1 105.134} C_DIS
LIN {X -0.167,Y -670.179,Z 1361.380,A 0.000,B 0.000,C 90.000,E1 104.411} C_DIS
LIN {X 0.345,Y -670.904,Z 1361.377,A 0.000,B 0.000,C 90.000,E1 103.883} C_DIS
LIN {X 0.146,Y -671.605,Z 1361.373,A 0.000,B 0.000,C 90.000,E1 103.175} C_DIS
LIN {X 0.017,Y -671.800,Z 1361.371,A 0.000,B 0.000,C 90.000,E1 102.703} C_DIS
LIN {X -0.257,Y -671.838,Z 1361.368,A 0.000,B 0.000,C 90.000,E1 102.243} C_DIS
LIN {X 0.208,Y -671.497,Z 1361.364,A 0.000,B 0.000,C 90.000,E1 101.478} C_DIS
LIN {X 0.074,Y -671.039,Z 1361.361,A 0.000,B 0.000,C 90.000,E1 101.007} C_DIS
LIN {X -0.190,Y -670.408,Z 1361.359,A 0.000,B 0.000,C 90.000,E1 100.546} C_DIS
LIN {X 0.134,Y -668.978,Z 1361.354,A 0.000,B 0.000,C 90.000,E1 99.792} C_DIS
LIN {X -0.024,Y -667.707,Z 1361.352,A 0.000,B 0.000,C 90.000,E1 99.321} C_DIS
LIN {X -0.298,Y -666.181,Z 1361.349,A 0.000,B 0.000,C 90.000,E1 98.859} C_DIS
LIN {X -0.017,Y -663.445,Z 1361.345,A 0.000,B 0.000,C 90.000,E1 98.106} C_DIS
LIN {X -0.312,Y -661.432,Z 1361.342,A 0.000,B 0.000,C 90.000,E1 97.644} C_DIS
LIN {X -0.082,Y -658.023,Z 1361.338,A 0.000,B 0.000,C 90.000,E1 96.891} C_DIS
LIN {X 0.241,Y -655.596,Z 1361.336,A 0.000,B 0.000,C 90.000,E1 96.372} C_DIS
LIN {X -0.107,Y -652.879,Z 1361.333,A 0.000,B 0.000,C 90.000,E1 95.910} C_DIS
LIN {X 0.064,Y -649.124,Z 1361.329,A 0.000,B 0.000,C 90.000,E1 95.277} C_DIS
LIN {X 0.089,Y -644.377,Z 1361.325,A 0.000,B 0.000,C 90.000,E1 94.531} C_DIS
LIN {X 0.188,Y -640.062,Z 1361.322,A 0.000,B 0.000,C 90.000,E1 93.898} C_DIS
LIN {X -0.301,Y -636.268,Z 1361.319,A 0.000,B 0.000,C 90.000,E1 93.440} C_DIS
LIN {X -0.272,Y -630.615,Z 1361.316,A 0.000,B 0.000,C 90.000,E1 92.808} C_DIS
LIN {X -0.196,Y -624.451,Z 1361.312,A 0.000,B 0.000,C 90.000,E1 92.178} C_DIS
LIN {X -0.195,Y -615.511,Z 1361.307,A 0.000,B 0.000,C 90.000,E1 91.318} C_DIS
LIN {X 0.190,Y -610.058,Z 1361.305,A 0.000,B 0.000,C 90.000,E1 90.802} C_DIS
LIN {X -0.239,Y -604.099,Z 1361.302,A 0.000,B 0.000,C 90.000,E1 90.401} C_DIS
LIN {X -0.163,Y -602.522,Z 1361.302,A 0.000,B 0.000,C 90.000,E1 90.286} C_DIS
LIN {X 0.038,Y -595.681,Z 1361.299,A 0.000,B 0.000,C 90.000,E1 89.885} C_DIS
LIN {X -0.227,Y -590.141,Z 1361.298,A 0.000,B 0.000,C 90.000,E1 89.656} C_DIS
LIN {X 0.197,Y -581.633,Z 1361.296,A 0.000,B 0.000,C 90.000,E1 89.255} C_DIS
LIN {X -0.215,Y -577.424,Z 1361.295,A 0.000,B 0.000,C 90.000,E1 89.083} C_DIS
LIN {X -0.175,Y -574.318,Z 1361.294,A 0.000,B 0.000,C 90.000,E1 88.854} C_DIS
LIN {X -0.208,Y -574.301,Z 1361.294,A 0.000,B 0.000,C 90.000,E1 88.854} C_DIS
LIN {X 0.054,Y -573.500,Z 1361.292,A 0.000,B 0.000,C 90.000,E1 88.625} C_DIS
LIN {X -0.019,Y -573.267,Z 1361.290,A 0.000,B 0.000,C 90.000,E1 88.224} C_DIS
LIN {X 0.014,Y -575.812,Z 1361.274,A 0.000,B 0.000,C 90.000,E1 85.241} C_DIS
LIN {X -0.128,Y -577.620,Z 1361.265,A 0.000,B 0.000,C 90.000,E1 83.628} C_DIS
LIN {X -0.021,Y -579.846,Z 1361.254,A 0.000,B 0.000,C 90.000,E1 81.724} C_DIS
LIN {X -0.143,Y -581.485,Z 1361.247,A 0.000,B 0.000,C 90.000,E1 80.387} C_DIS
LIN {X -0.235,Y -582.942,Z 1361.239,A 0.000,B 0.000,C 90.000,E1 79.050} C_DIS
LIN {X 0.142,Y -584.024,Z 1361.233,A 0.000,B 0.000,C 90.000,E1 77.937} C_DIS
LIN {X 0.121,Y -585.741,Z 1361.223,A 0.000,B 0.000,C 90.000,E1 76.061} C_DIS
LIN {X 0.180,Y -586.933,Z 1361.214,A 0.000,B 0.000,C 90.000,E1 74.448} C_DIS
LIN {X 0.197,Y -588.278,Z 1361.202,A 0.000,B 0.000,C 90.000,E1 72.308} C_DIS
LIN {X 0.256,Y -589.004,Z 1361.194,A 0.000,B 0.000,C 90.000,E1 70.967} C_DIS
LIN {X 0.134,Y -589.786,Z 1361.187,A 0.000,B 0.000,C 90.000,E1 69.645} C_DIS
LIN {X -0.015,Y -590.948,Z 1361.177,A 0.000,B 0.000,C 90.000,E1 67.794} C_DIS
LIN {X 0.098,Y -592.300,Z 1361.166,A 0.000,B 0.000,C 90.000,E1 65.921} C_DIS
LIN {X 0.146,Y -593.461,Z 1361.159,A 0.000,B 0.000,C 90.000,E1 64.588} C_DIS
LIN {X 0.122,Y -594.636,Z 1361.150,A 0.000,B 0.000,C 90.000,E1 62.999} C_DIS
LIN {X -0.225,Y -596.090,Z 1361.140,A 0.000,B 0.000,C 90.000,E1 61.179} C_DIS
LIN {X -0.197,Y -596.787,Z 1361.135,A 0.000,B 0.000,C 90.000,E1 60.383} C_DIS
LIN {X -0.159,Y -597.572,Z 1361.131,A 0.000,B 0.000,C 90.000,E1 59.587} C_DIS
LIN {X -0.202,Y -598.623,Z 1361.125,A 0.000,B 0.000,C 90.000,E1 58.535} C_DIS
LIN {X 0.222,Y -600.161,Z 1361.116,A 0.000,B 0.000,C 90.000,E1 56.914} C_DIS
LIN {X 0.017,Y -601.137,Z 1361.110,A 0.000,B 0.000,C 90.000,E1 55.881} C_DIS
LIN {X 0.087,Y -602.807,Z 1361.100,A 0.000,B 0.000,C 90.000,E1 54.036} C_DIS
LIN {X 0.012,Y -603.586,Z 1361.096,A 0.000,B 0.000,C 90.000,E1 53.256} C_DIS
LIN {X 0.203,Y -604.474,Z 1361.090,A 0.000,B 0.000,C 90.000,E1 52.190} C_DIS
LIN {X 0.184,Y -605.358,Z 1361.083,A 0.000,B 0.000,C 90.000,E1 50.884} C_DIS
LIN {X 0.098,Y -606.122,Z 1361.076,A 0.000,B 0.000,C 90.000,E1 49.585} C_DIS
LIN {X -0.173,Y -606.623,Z 1361.070,A 0.000,B 0.000,C 90.000,E1 48.566} C_DIS
LIN {X 0.168,Y -606.964,Z 1361.063,A 0.000,B 0.000,C 90.000,E1 47.229} C_DIS
LIN {X -0.338,Y -607.117,Z 1361.055,A 0.000,B 0.000,C 90.000,E1 45.972} C_DIS
LIN {X -0.232,Y -607.127,Z 1361.049,A 0.000,B 0.000,C 90.000,E1 44.919} C_DIS
LIN {X -0.127,Y -606.917,Z 1361.044,A 0.000,B 0.000,C 90.000,E1 43.866} C_DIS
LIN {X -0.032,Y -606.495,Z 1361.038,A 0.000,B 0.000,C 90.000,E1 42.813} C_DIS
LIN {X 0.151,Y -605.780,Z 1361.029,A 0.000,B 0.000,C 90.000,E1 41.229} C_DIS
LIN {X 0.012,Y -605.341,Z 1361.025,A 0.000,B 0.000,C 90.000,E1 40.458} C_DIS
LIN {X 0.120,Y -604.717,Z 1361.019,A 0.000,B 0.000,C 90.000,E1 39.402} C_DIS
LIN {X 0.097,Y -603.768,Z 1361.012,A 0.000,B 0.000,C 90.000,E1 38.096} C_DIS
LIN {X 0.026,Y -603.085,Z 1361.007,A 0.000,B 0.000,C 90.000,E1 37.317} C_DIS
LIN {X -0.277,Y -601.943,Z 1361.002,A 0.000,B 0.000,C 90.000,E1 36.297} C_DIS
LIN {X -0.116,Y -600.278,Z 1360.996,A 0.000,B 0.000,C 90.000,E1 35.231} C_DIS
LIN {X 0.028,Y -599.369,Z 1360.993,A 0.000,B 0.000,C 90.000,E1 34.692} C_DIS
LIN {X 0.144,Y -597.128,Z 1360.987,A 0.000,B 0.000,C 90.000,E1 33.627} C_DIS
LIN {X -0.214,Y -594.001,Z 1360.980,A 0.000,B 0.000,C 90.000,E1 32.339} C_DIS
LIN {X -0.211,Y -591.688,Z 1360.975,A 0.000,B 0.000,C 90.000,E1 31.544} C_DIS
LIN {X -0.037,Y -588.184,Z 1360.969,A 0.000,B 0.000,C 90.000,E1 30.463} C_DIS
LIN {X -0.092,Y -585.133,Z 1360.965,A 0.000,B 0.000,C 90.000,E1 29.667} C_DIS
LIN {X -0.179,Y -581.804,Z 1360.960,A 0.000,B 0.000,C 90.000,E1 28.871} C_DIS
LIN {X 0.068,Y -579.292,Z 1360.957,A 0.000,B 0.000,C 90.000,E1 28.309} C_DIS
LIN {X -0.165,Y -574.569,Z 1360.952,A 0.000,B 0.000,C 90.000,E1 27.385} C_DIS
LIN {X -0.044,Y -570.900,Z 1360.948,A 0.000,B 0.000,C 90.000,E1 26.693} C_DIS
LIN {X -0.124,Y -567.736,Z 1360.945,A 0.000,B 0.000,C 90.000,E1 26.155} C_DIS
LIN {X -0.064,Y -563.487,Z 1360.942,A 0.000,B 0.000,C 90.000,E1 25.463} C_DIS
LIN {X -0.038,Y -558.980,Z 1360.938,A 0.000,B 0.000,C 90.000,E1 24.771} C_DIS
LIN {X -0.053,Y -553.963,Z 1360.934,A 0.000,B 0.000,C 90.000,E1 24.079} C_DIS
LIN {X 0.153,Y -546.432,Z 1360.928,A 0.000,B 0.000,C 90.000,E1 23.078} C_DIS
LIN {X 0.051,Y -538.161,Z 1360.923,A 0.000,B 0.000,C 90.000,E1 22.099} C_DIS
LIN {X -0.007,Y -533.182,Z 1360.920,A 0.000,B 0.000,C 90.000,E1 21.535} C_DIS
LIN {X 0.061,Y -524.256,Z 1360.914,A 0.000,B 0.000,C 90.000,E1 20.556} C_DIS
LIN {X 0.037,Y -513.675,Z 1360.908,A 0.000,B 0.000,C 90.000,E1 19.450} C_DIS
LIN {X 0.098,Y -501.525,Z 1360.901,A 0.000,B 0.000,C 90.000,E1 18.181} C_DIS
LIN {X 0.111,Y -493.350,Z 1360.896,A 0.000,B 0.000,C 90.000,E1 17.330} C_DIS
LIN {X 0.083,Y -482.160,Z 1360.890,A 0.000,B 0.000,C 90.000,E1 16.260} C_DIS
LIN {X -0.189,Y -466.672,Z 1360.882,A 0.000,B 0.000,C 90.000,E1 14.773} C_DIS
LIN {X -0.007,Y -453.830,Z 1360.875,A 0.000,B 0.000,C 90.000,E1 13.480} C_DIS
LIN {X 0.114,Y -436.830,Z 1360.865,A 0.000,B 0.000,C 90.000,E1 11.715} C_DIS
LIN {X 0.152,Y -419.992,Z 1360.855,A 0.000,B 0.000,C 90.000,E1 9.849} C_DIS
LIN {X -0.120,Y -405.940,Z 1360.846,A 0.000,B 0.000,C 90.000,E1 8.276} C_DIS
LIN {X -0.186,Y -397.442,Z 1360.840,A 0.000,B 0.000,C 90.000,E1 7.296} C_DIS
LIN {X -0.068,Y -393.239,Z 1360.837,A 0.000,B 0.000,C 90.000,E1 6.663} C_DIS
LIN {X -0.106,Y -393.244,Z 1360.837,A 0.000,B 0.000,C 90.000,E1 6.663} C_DIS
LIN {X -0.014,Y -394.528,Z 1360.836,A 0.000,B 0.000,C 90.000,E1 6.429} C_DIS
LIN {X -0.015,Y -398.891,Z 1360.833,A 0.000,B 0.000,C 90.000,E1 6.030} C_DIS
LIN {X -0.086,Y -409.704,Z 1360.829,A 0.000,B 0.000,C 90.000,E1 5.277} C_DIS
LIN {X 0.116,Y -415.864,Z 1360.827,A 0.000,B 0.000,C 90.000,E1 4.759} C_DIS
LIN {X 0.124,Y -420.426,Z 1360.824,A 0.000,B 0.000,C 90.000,E1 4.359} C_DIS
LIN {X 0.163,Y -423.401,Z 1360.823,A 0.000,B 0.000,C 90.000,E1 4.073} C_DIS
LIN {X 0.116,Y -430.437,Z 1360.819,A 0.000,B 0.000,C 90.000,E1 3.326} C_DIS
LIN {X 0.130,Y -435.887,Z 1360.815,A 0.000,B 0.000,C 90.000,E1 2.694} C_DIS
LIN {X 0.065,Y -443.433,Z 1360.810,A 0.000,B 0.000,C 90.000,E1 1.776} C_DIS
LIN {X -0.185,Y -449.451,Z 1360.806,A 0.000,B 0.000,C 90.000,E1 1.031} C_DIS
LIN {X 0.211,Y -455.283,Z 1360.801,A 0.000,B 0.000,C 90.000,E1 0.172} C_DIS
LIN {X 0.001,Y -461.276,Z 1360.796,A 0.000,B 0.000,C 90.000,E1 359.312} C_DIS
LIN {X 0.058,Y -466.332,Z 1360.792,A 0.000,B 0.000,C 90.000,E1 358.511} C_DIS
LIN {X 0.181,Y -471.008,Z 1360.787,A 0.000,B 0.000,C 90.000,E1 357.707} C_DIS
LIN {X -0.144,Y -475.283,Z 1360.783,A 0.000,B 0.000,C 90.000,E1 356.963} C_DIS
LIN {X 0.069,Y -479.311,Z 1360.779,A 0.000,B 0.000,C 90.000,E1 356.159} C_DIS
LIN {X -0.159,Y -482.954,Z 1360.774,A 0.000,B 0.000,C 90.000,E1 355.412} C_DIS
LIN {X 0.131,Y -486.315,Z 1360.770,A 0.000,B 0.000,C 90.000,E1 354.609} C_DIS
LIN {X 0.143,Y -488.247,Z 1360.768,A 0.000,B 0.000,C 90.000,E1 354.147} C_DIS
LIN {X 0.203,Y -491.662,Z 1360.763,A 0.000,B 0.000,C 90.000,E1 353.223} C_DIS
LIN {X -0.083,Y -493.780,Z 1360.759,A 0.000,B 0.000,C 90.000,E1 352.648} C_DIS
LIN {X 0.036,Y -496.549,Z 1360.754,A 0.000,B 0.000,C 90.000,E1 351.724} C_DIS
LIN {X 0.261,Y -499.047,Z 1360.749,A 0.000,B 0.000,C 90.000,E1 350.792} C_DIS
LIN {X -0.058,Y -501.416,Z 1360.744,A 0.000,B 0.000,C 90.000,E1 349.926} C_DIS
LIN {X -0.201,Y -502.859,Z 1360.741,A 0.000,B 0.000,C 90.000,E1 349.342} C_DIS
LIN {X 0.099,Y -504.715,Z 1360.736,A 0.000,B 0.000,C 90.000,E1 348.409} C_DIS
LIN {X -0.019,Y -506.976,Z 1360.729,A 0.000,B 0.000,C 90.000,E1 347.229} C_DIS
LIN {X -0.140,Y -509.256,Z 1360.721,A 0.000,B 0.000,C 90.000,E1 345.755} C_DIS
LIN {X -0.144,Y -510.285,Z 1360.716,A 0.000,B 0.000,C 90.000,E1 344.866} C_DIS
LIN {X -0.137,Y -511.139,Z 1360.711,A 0.000,B 0.000,C 90.000,E1 343.976} C_DIS
LIN {X -0.181,Y -511.366,Z 1360.709,A 0.000,B 0.000,C 90.000,E1 343.685} C_DIS
LIN {X -0.080,Y -511.421,Z 1360.708,A 0.000,B 0.000,C 90.000,E1 343.378} C_DIS
LIN {X -0.124,Y -511.342,Z 1360.706,A 0.000,B 0.000,C 90.000,E1 343.087} C_DIS
LIN {X -0.020,Y -511.052,Z 1360.704,A 0.000,B 0.000,C 90.000,E1 342.779} C_DIS
LIN {X -0.067,Y -510.412,Z 1360.703,A 0.000,B 0.000,C 90.000,E1 342.489} C_DIS
LIN {X 0.037,Y -509.201,Z 1360.701,A 0.000,B 0.000,C 90.000,E1 342.181} C_DIS
LIN {X -0.153,Y -507.873,Z 1360.700,A 0.000,B 0.000,C 90.000,E1 342.054} C_DIS
LIN {X -0.044,Y -497.134,Z 1360.698,A 0.000,B 0.000,C 90.000,E1 341.638} C_DIS
LIN {X 0.145,Y -466.182,Z 1360.691,A 0.000,B 0.000,C 90.000,E1 340.369} C_DIS
LIN {X 0.013,Y -438.903,Z 1360.684,A 0.000,B 0.000,C 90.000,E1 339.135} C_DIS
LIN {X 0.164,Y -413.514,Z 1360.677,A 0.000,B 0.000,C 90.000,E1 337.794} C_DIS
LIN {X -0.003,Y -390.019,Z 1360.669,A 0.000,B 0.000,C 90.000,E1 336.433} C_DIS
LIN {X 0.139,Y -368.456,Z 1360.661,A 0.000,B 0.000,C 90.000,E1 334.973} C_DIS
LIN {X -0.120,Y -363.612,Z 1360.659,A 0.000,B 0.000,C 90.000,E1 334.665} C_DIS
LIN {X -0.144,Y -363.599,Z 1360.659,A 0.000,B 0.000,C 90.000,E1 334.665} C_DIS
LIN {X 0.166,Y -366.109,Z 1360.642,A 0.000,B 0.000,C 90.000,E1 331.513} C_DIS
LIN {X -0.112,Y -370.670,Z 1360.607,A 0.000,B 0.000,C 90.000,E1 325.261} C_DIS
LIN {X 0.161,Y -371.508,Z 1360.603,A 0.000,B 0.000,C 90.000,E1 324.482} C_DIS
LIN {X -0.077,Y -372.046,Z 1360.599,A 0.000,B 0.000,C 90.000,E1 323.783} C_DIS
LIN {X -0.038,Y -378.005,Z 1360.564,A 0.000,B 0.000,C 90.000,E1 317.553} C_DIS
LIN {X 0.000,Y -379.381,Z 1360.554,A 0.000,B 0.000,C 90.000,E1 315.729} C_DIS
LIN {X 0.021,Y -384.613,Z 1360.528,A 0.000,B 0.000,C 90.000,E1 311.024} C_DIS
LIN {X 0.073,Y -385.220,Z 1360.524,A 0.000,B 0.000,C 90.000,E1 310.297} C_DIS
LIN {X -0.210,Y -391.271,Z 1360.492,A 0.000,B 0.000,C 90.000,E1 304.612} C_DIS
LIN {X -0.057,Y -396.984,Z 1360.459,A 0.000,B 0.000,C 90.000,E1 298.565} C_DIS
LIN {X -0.106,Y -401.349,Z 1360.427,A 0.000,B 0.000,C 90.000,E1 292.950} C_DIS
LIN {X -0.026,Y -401.658,Z 1360.426,A 0.000,B 0.000,C 90.000,E1 292.589} C_DIS
LIN {X 0.127,Y -404.748,Z 1360.395,A 0.000,B 0.000,C 90.000,E1 286.985} C_DIS
LIN {X 0.140,Y -406.156,Z 1360.364,A 0.000,B 0.000,C 90.000,E1 281.422} C_DIS
LIN {X -0.159,Y -405.677,Z 1360.333,A 0.000,B 0.000,C 90.000,E1 275.910} C_DIS
LIN {X -0.088,Y -403.565,Z 1360.306,A 0.000,B 0.000,C 90.000,E1 271.031} C_DIS
LIN {X -0.153,Y -403.174,Z 1360.302,A 0.000,B 0.000,C 90.000,E1 270.344} C_DIS
LIN {X 0.081,Y -399.064,Z 1360.273,A 0.000,B 0.000,C 90.000,E1 265.065} C_DIS
LIN {X 0.022,Y -398.767,Z 1360.271,A 0.000,B 0.000,C 90.000,E1 264.723} C_DIS
LIN {X -0.088,Y -393.287,Z 1360.243,A 0.000,B 0.000,C 90.000,E1 259.803} C_DIS
LIN {X -0.167,Y -392.661,Z 1360.239,A 0.000,B 0.000,C 90.000,E1 259.106} C_DIS
LIN {X 0.003,Y -386.241,Z 1360.214,A 0.000,B 0.000,C 90.000,E1 254.448} C_DIS
LIN {X -0.031,Y -385.144,Z 1360.208,A 0.000,B 0.000,C 90.000,E1 253.378} C_DIS
LIN {X 0.077,Y -377.808,Z 1360.182,A 0.000,B 0.000,C 90.000,E1 248.666} C_DIS
LIN {X -0.051,Y -376.076,Z 1360.173,A 0.000,B 0.000,C 90.000,E1 247.230} C_DIS
LIN {X 0.007,Y -368.744,Z 1360.149,A 0.000,B 0.000,C 90.000,E1 242.820} C_DIS
LIN {X -0.008,Y -366.391,Z 1360.139,A 0.000,B 0.000,C 90.000,E1 240.973} C_DIS
LIN {X 0.157,Y -365.091,Z 1360.135,A 0.000,B 0.000,C 90.000,E1 240.205} C_DIS
LIN {X -0.094,Y -358.496,Z 1360.112,A 0.000,B 0.000,C 90.000,E1 236.135} C_DIS
LIN {X -0.034,Y -356.171,Z 1360.101,A 0.000,B 0.000,C 90.000,E1 234.242} C_DIS
LIN {X -0.095,Y -354.922,Z 1360.097,A 0.000,B 0.000,C 90.000,E1 233.497} C_DIS
LIN {X -0.111,Y -348.153,Z 1360.072,A 0.000,B 0.000,C 90.000,E1 228.933} C_DIS
LIN {X 0.060,Y -346.050,Z 1360.061,A 0.000,B 0.000,C 90.000,E1 226.986} C_DIS
LIN {X 0.032,Y -339.249,Z 1360.033,A 0.000,B 0.000,C 90.000,E1 221.962} C_DIS
LIN {X -0.032,Y -336.660,Z 1360.018,A 0.000,B 0.000,C 90.000,E1 219.241} C_DIS
LIN {X 0.125,Y -330.753,Z 1359.987,A 0.000,B 0.000,C 90.000,E1 213.706} C_DIS
LIN {X 0.077,Y -329.194,Z 1359.974,A 0.000,B 0.000,C 90.000,E1 211.337} C_DIS
LIN {X -0.045,Y -326.784,Z 1359.960,A 0.000,B 0.000,C 90.000,E1 208.821} C_DIS
LIN {X -0.062,Y -326.782,Z 1359.960,A 0.000,B 0.000,C 90.000,E1 208.821} C_DIS
LIN {X 0.058,Y -344.297,Z 1359.952,A 0.000,B 0.000,C 90.000,E1 207.257} C_DIS
LIN {X -0.157,Y -364.399,Z 1359.943,A 0.000,B 0.000,C 90.000,E1 205.720} C_DIS
LIN {X 0.126,Y -386.454,Z 1359.934,A 0.000,B 0.000,C 90.000,E1 204.155} C_DIS
LIN {X -0.010,Y -410.459,Z 1359.926,A 0.000,B 0.000,C 90.000,E1 202.717} C_DIS
LIN {X -0.031,Y -436.422,Z 1359.919,A 0.000,B 0.000,C 90.000,E1 201.334} C_DIS
LIN {X -0.123,Y -445.135,Z 1359.916,A 0.000,B 0.000,C 90.000,E1 200.918} C_DIS
LIN {X -0.007,Y -448.038,Z 1359.915,A 0.000,B 0.000,C 90.000,E1 200.737} C_DIS
LIN {X -0.100,Y -449.409,Z 1359.914,A 0.000,B 0.000,C 90.000,E1 200.556} C_DIS
LIN {X 0.048,Y -450.159,Z 1359.913,A 0.000,B 0.000,C 90.000,E1 200.375} C_DIS
LIN {X -0.226,Y -450.751,Z 1359.912,A 0.000,B 0.000,C 90.000,E1 200.248} C_DIS
LIN {X 0.079,Y -451.669,Z 1359.911,A 0.000,B 0.000,C 90.000,E1 199.885} C_DIS
LIN {X -0.037,Y -452.370,Z 1359.909,A 0.000,B 0.000,C 90.000,E1 199.577} C_DIS
LIN {X 0.164,Y -453.265,Z 1359.905,A 0.000,B 0.000,C 90.000,E1 198.906} C_DIS
LIN {X 0.090,Y -454.987,Z 1359.895,A 0.000,B 0.000,C 90.000,E1 196.985} C_DIS
LIN {X 0.160,Y -456.231,Z 1359.885,A 0.000,B 0.000,C 90.000,E1 195.371} C_DIS
LIN {X 0.132,Y -457.411,Z 1359.877,A 0.000,B 0.000,C 90.000,E1 193.772} C_DIS
LIN {X 0.021,Y -458.547,Z 1359.868,A 0.000,B 0.000,C 90.000,E1 192.187} C_DIS
LIN {X -0.074,Y -459.654,Z 1359.859,A 0.000,B 0.000,C 90.000,E1 190.602} C_DIS
LIN {X 0.211,Y -460.584,Z 1359.850,A 0.000,B 0.000,C 90.000,E1 188.973} C_DIS
LIN {X -0.017,Y -461.327,Z 1359.841,A 0.000,B 0.000,C 90.000,E1 187.409} C_DIS
LIN {X 0.166,Y -461.762,Z 1359.832,A 0.000,B 0.000,C 90.000,E1 185.796} C_DIS
LIN {X -0.119,Y -461.915,Z 1359.827,A 0.000,B 0.000,C 90.000,E1 184.878} C_DIS
LIN {X -0.163,Y -461.951,Z 1359.820,A 0.000,B 0.000,C 90.000,E1 183.612} C_DIS
LIN {X 0.018,Y -461.860,Z 1359.815,A 0.000,B 0.000,C 90.000,E1 182.636} C_DIS
LIN {X -0.062,Y -461.488,Z 1359.808,A 0.000,B 0.000,C 90.000,E1 181.375} C_DIS
LIN {X 0.098,Y -460.930,Z 1359.802,A 0.000,B 0.000,C 90.000,E1 180.401} C_DIS
LIN {X 0.047,Y -460.303,Z 1359.799,A 0.000,B 0.000,C 90.000,E1 179.771} C_DIS
LIN {X 0.192,Y -459.052,Z 1359.793,A 0.000,B 0.000,C 90.000,E1 178.797} C_DIS
LIN {X -0.124,Y -457.561,Z 1359.788,A 0.000,B 0.000,C 90.000,E1 177.879} C_DIS
LIN {X -0.201,Y -456.381,Z 1359.785,A 0.000,B 0.000,C 90.000,E1 177.249} C_DIS
LIN {X -0.088,Y -453.832,Z 1359.779,A 0.000,B 0.000,C 90.000,E1 176.274} C_DIS
LIN {X -0.169,Y -452.010,Z 1359.776,A 0.000,B 0.000,C 90.000,E1 175.641} C_DIS
LIN {X 0.186,Y -449.806,Z 1359.772,A 0.000,B 0.000,C 90.000,E1 174.951} C_DIS
LIN {X -0.123,Y -445.096,Z 1359.766,A 0.000,B 0.000,C 90.000,E1 173.856} C_DIS
LIN {X -0.110,Y -440.036,Z 1359.760,A 0.000,B 0.000,C 90.000,E1 172.875} C_DIS
LIN {X 0.135,Y -436.223,Z 1359.757,A 0.000,B 0.000,C 90.000,E1 172.186} C_DIS
LIN {X 0.006,Y -430.851,Z 1359.752,A 0.000,B 0.000,C 90.000,E1 171.376} C_DIS
LIN {X -0.192,Y -426.218,Z 1359.748,A 0.000,B 0.000,C 90.000,E1 170.735} C_DIS
LIN {X -0.095,Y -411.259,Z 1359.736,A 0.000,B 0.000,C 90.000,E1 168.522} C_DIS
LIN {X 0.146,Y -398.377,Z 1359.725,A 0.000,B 0.000,C 90.000,E1 166.408} C_DIS
LIN {X 0.184,Y -397.410,Z 1359.724,A 0.000,B 0.000,C 90.000,E1 166.228} C_DIS
LIN {X -0.020,Y -394.519,Z 1359.720,A 0.000,B 0.000,C 90.000,E1 165.589} C_DIS
LIN {X 0.008,Y -393.879,Z 1359.719,A 0.000,B 0.000,C 90.000,E1 165.408} C_DIS
LIN {X -0.083,Y -393.214,Z 1359.717,A 0.000,B 0.000,C 90.000,E1 164.991} C_DIS
LIN {X -0.057,Y -393.348,Z 1359.716,A 0.000,B 0.000,C 90.000,E1 164.810} C_DIS
LIN {X -0.004,Y -394.830,Z 1359.714,A 0.000,B 0.000,C 90.000,E1 164.448} C_DIS
LIN {X -0.041,Y -397.479,Z 1359.712,A 0.000,B 0.000,C 90.000,E1 164.102} C_DIS
LIN {X 0.003,Y -398.712,Z 1359.711,A 0.000,B 0.000,C 90.000,E1 163.921} C_DIS
LIN {X -0.133,Y -405.015,Z 1359.707,A 0.000,B 0.000,C 90.000,E1 163.251} C_DIS
LIN {X -0.018,Y -413.843,Z 1359.702,A 0.000,B 0.000,C 90.000,E1 162.417} C_DIS
LIN {X -0.049,Y -434.367,Z 1359.693,A 0.000,B 0.000,C 90.000,E1 160.732} C_DIS
LIN {X 0.195,Y -453.263,Z 1359.685,A 0.000,B 0.000,C 90.000,E1 159.263} C_DIS
LIN {X -0.096,Y -459.441,Z 1359.682,A 0.000,B 0.000,C 90.000,E1 158.827} C_DIS
LIN {X -0.165,Y -466.998,Z 1359.679,A 0.000,B 0.000,C 90.000,E1 158.230} C_DIS
LIN {X -0.118,Y -473.049,Z 1359.676,A 0.000,B 0.000,C 90.000,E1 157.720} C_DIS
LIN {X 0.096,Y -478.997,Z 1359.673,A 0.000,B 0.000,C 90.000,E1 157.177} C_DIS
LIN {X -0.024,Y -484.868,Z 1359.670,A 0.000,B 0.000,C 90.000,E1 156.666} C_DIS
LIN {X -0.115,Y -493.467,Z 1359.666,A 0.000,B 0.000,C 90.000,E1 155.869} C_DIS
LIN {X -0.171,Y -501.690,Z 1359.661,A 0.000,B 0.000,C 90.000,E1 155.049} C_DIS
LIN {X 0.214,Y -505.628,Z 1359.659,A 0.000,B 0.000,C 90.000,E1 154.588} C_DIS
LIN {X 0.100,Y -510.773,Z 1359.656,A 0.000,B 0.000,C 90.000,E1 154.024} C_DIS
LIN {X -0.093,Y -517.015,Z 1359.652,A 0.000,B 0.000,C 90.000,E1 153.307} C_DIS
LIN {X -0.009,Y -522.635,Z 1359.648,A 0.000,B 0.000,C 90.000,E1 152.564} C_DIS
LIN {X 0.055,Y -526.697,Z 1359.644,A 0.000,B 0.000,C 90.000,E1 151.975} C_DIS
LIN {X 0.154,Y -530.351,Z 1359.641,A 0.000,B 0.000,C 90.000,E1 151.385} C_DIS
LIN {X 0.134,Y -534.029,Z 1359.637,A 0.000,B 0.000,C 90.000,E1 150.667} C_DIS
LIN {X -0.179,Y -536.652,Z 1359.634,A 0.000,B 0.000,C 90.000,E1 150.127} C_DIS
LIN {X 0.133,Y -538.385,Z 1359.632,A 0.000,B 0.000,C 90.000,E1 149.665} C_DIS
LIN {X 0.038,Y -541.364,Z 1359.627,A 0.000,B 0.000,C 90.000,E1 148.820} C_DIS
LIN {X 0.059,Y -543.142,Z 1359.624,A 0.000,B 0.000,C 90.000,E1 148.250} C_DIS
LIN {X 0.004,Y -545.318,Z 1359.619,A 0.000,B 0.000,C 90.000,E1 147.406} C_DIS
LIN {X 0.103,Y -547.048,Z 1359.614,A 0.000,B 0.000,C 90.000,E1 146.548} C_DIS
LIN {X -0.075,Y -548.551,Z 1359.610,A 0.000,B 0.000,C 90.000,E1 145.722} C_DIS
LIN {X -0.290,Y -549.435,Z 1359.606,A 0.000,B 0.000,C 90.000,E1 145.182} C_DIS
LIN {X -0.130,Y -550.503,Z 1359.602,A 0.000,B 0.000,C 90.000,E1 144.322} C_DIS
LIN {X -0.281,Y -551.426,Z 1359.597,A 0.000,B 0.000,C 90.000,E1 143.497} C_DIS
LIN {X -0.036,Y -552.393,Z 1359.591,A 0.000,B 0.000,C 90.000,E1 142.351} C_DIS
LIN {X -0.215,Y -553.206,Z 1359.585,A 0.000,B 0.000,C 90.000,E1 141.251} C_DIS
LIN {X 0.039,Y -554.108,Z 1359.577,A 0.000,B 0.000,C 90.000,E1 139.828} C_DIS
LIN {X -0.106,Y -554.982,Z 1359.569,A 0.000,B 0.000,C 90.000,E1 138.447} C_DIS
LIN {X -0.177,Y -555.805,Z 1359.560,A 0.000,B 0.000,C 90.000,E1 136.782} C_DIS
LIN {X 0.072,Y -556.394,Z 1359.552,A 0.000,B 0.000,C 90.000,E1 135.364} C_DIS
LIN {X 0.055,Y -557.378,Z 1359.541,A 0.000,B 0.000,C 90.000,E1 133.419} C_DIS
LIN {X -0.105,Y -558.266,Z 1359.535,A 0.000,B 0.000,C 90.000,E1 132.324} C_DIS
LIN {X 0.011,Y -559.221,Z 1359.532,A 0.000,B 0.000,C 90.000,E1 131.757} C_DIS
LIN {X -0.107,Y -559.885,Z 1359.531,A 0.000,B 0.000,C 90.000,E1 131.553} C_DIS
LIN {X 0.222,Y -559.921,Z 1359.531,A 0.000,B 0.000,C 90.000,E1 131.515} C_DIS
LIN {X 0.091,Y -560.759,Z 1359.531,A 0.000,B 0.000,C 90.000,E1 131.472} C_DIS
LIN {X -0.127,Y -562.977,Z 1359.530,A 0.000,B 0.000,C 90.000,E1 131.391} C_DIS
LIN {X -0.058,Y -573.270,Z 1359.528,A 0.000,B 0.000,C 90.000,E1 131.067} C_DIS
LIN {X 0.091,Y -579.969,Z 1359.527,A 0.000,B 0.000,C 90.000,E1 130.825} C_DIS
LIN {X 0.123,Y -585.669,Z 1359.525,A 0.000,B 0.000,C 90.000,E1 130.539} C_DIS
LIN {X 0.290,Y -591.449,Z 1359.523,A 0.000,B 0.000,C 90.000,E1 130.172} C_DIS
LIN {X -0.101,Y -595.609,Z 1359.522,A 0.000,B 0.000,C 90.000,E1 129.930} C_DIS
LIN {X -0.338,Y -599.780,Z 1359.520,A 0.000,B 0.000,C 90.000,E1 129.644} C_DIS
LIN {X -0.016,Y -603.923,Z 1359.518,A 0.000,B 0.000,C 90.000,E1 129.277} C_DIS
LIN {X 0.253,Y -611.671,Z 1359.514,A 0.000,B 0.000,C 90.000,E1 128.543} C_DIS
LIN {X -0.132,Y -616.572,Z 1359.512,A 0.000,B 0.000,C 90.000,E1 128.096} C_DIS
LIN {X 0.029,Y -621.212,Z 1359.509,A 0.000,B 0.000,C 90.000,E1 127.604} C_DIS
LIN {X 0.214,Y -627.049,Z 1359.505,A 0.000,B 0.000,C 90.000,E1 126.950} C_DIS
LIN {X 0.406,Y -632.542,Z 1359.502,A 0.000,B 0.000,C 90.000,E1 126.297} C_DIS
LIN {X -0.142,Y -637.725,Z 1359.498,A 0.000,B 0.000,C 90.000,E1 125.724} C_DIS
LIN {X 0.148,Y -643.625,Z 1359.494,A 0.000,B 0.000,C 90.000,E1 124.945} C_DIS
LIN {X 0.164,Y -649.869,Z 1359.489,A 0.000,B 0.000,C 90.000,E1 124.072} C_DIS
LIN {X -0.313,Y -654.772,Z 1359.485,A 0.000,B 0.000,C 90.000,E1 123.372} C_DIS
LIN {X -0.269,Y -658.440,Z 1359.482,A 0.000,B 0.000,C 90.000,E1 122.752} C_DIS
LIN {X -0.096,Y -662.141,Z 1359.478,A 0.000,B 0.000,C 90.000,E1 122.005} C_DIS
LIN {X -0.063,Y -664.448,Z 1359.475,A 0.000,B 0.000,C 90.000,E1 121.514} C_DIS
LIN {X -0.225,Y -667.434,Z 1359.471,A 0.000,B 0.000,C 90.000,E1 120.797} C_DIS
LIN {X -0.015,Y -669.825,Z 1359.467,A 0.000,B 0.000,C 90.000,E1 120.050} C_DIS
LIN {X 0.047,Y -672.417,Z 1359.462,A 0.000,B 0.000,C 90.000,E1 119.077} C_DIS
LIN {X -0.027,Y -673.529,Z 1359.458,A 0.000,B 0.000,C 90.000,E1 118.359} C_DIS
LIN {X -0.093,Y -673.958,Z 1359.454,A 0.000,B 0.000,C 90.000,E1 117.641} C_DIS
LIN {X -0.156,Y -673.939,Z 1359.450,A 0.000,B 0.000,C 90.000,E1 116.924} C_DIS
LIN {X -0.345,Y -673.541,Z 1359.444,A 0.000,B 0.000,C 90.000,E1 115.976} C_DIS
LIN {X 0.186,Y -672.938,Z 1359.440,A 0.000,B 0.000,C 90.000,E1 115.207} C_DIS
LIN {X -0.358,Y -672.252,Z 1359.438,A 0.000,B 0.000,C 90.000,E1 114.771} C_DIS
LIN {X -0.185,Y -671.706,Z 1359.436,A 0.000,B 0.000,C 90.000,E1 114.515} C_DIS
LIN {X -0.120,Y -670.184,Z 1359.433,A 0.000,B 0.000,C 90.000,E1 114.027} C_DIS
LIN {X -0.036,Y -669.555,Z 1359.433,A 0.000,B 0.000,C 90.000,E1 113.898} C_DIS
LIN {X 0.283,Y -666.306,Z 1359.430,A 0.000,B 0.000,C 90.000,E1 113.387} C_DIS
LIN {X 0.358,Y -665.200,Z 1359.429,A 0.000,B 0.000,C 90.000,E1 113.259} C_DIS
LIN {X 0.201,Y -659.168,Z 1359.427,A 0.000,B 0.000,C 90.000,E1 112.823} C_DIS
LIN {X 0.214,Y -657.238,Z 1359.426,A 0.000,B 0.000,C 90.000,E1 112.717} C_DIS
LIN {X -0.243,Y -652.532,Z 1359.425,A 0.000,B 0.000,C 90.000,E1 112.589} C_DIS
LIN {X 0.063,Y -647.149,Z 1359.424,A 0.000,B 0.000,C 90.000,E1 112.386} C_DIS
LIN {X -0.018,Y -642.650,Z 1359.424,A 0.000,B 0.000,C 90.000,E1 112.280} C_DIS
LIN {X 0.173,Y -632.463,Z 1359.422,A 0.000,B 0.000,C 90.000,E1 112.025} C_DIS
LIN {X 0.114,Y -632.482,Z 1359.422,A 0.000,B 0.000,C 90.000,E1 112.025} C_DIS
LIN {X 0.239,Y -637.932,Z 1359.419,A 0.000,B 0.000,C 90.000,E1 111.354} C_DIS
LIN {X 0.329,Y -644.265,Z 1359.415,A 0.000,B 0.000,C 90.000,E1 110.610} C_DIS
LIN {X 0.258,Y -648.761,Z 1359.411,A 0.000,B 0.000,C 90.000,E1 109.993} C_DIS
LIN {X 0.002,Y -652.374,Z 1359.408,A 0.000,B 0.000,C 90.000,E1 109.396} C_DIS
LIN {X -0.010,Y -655.542,Z 1359.404,A 0.000,B 0.000,C 90.000,E1 108.779} C_DIS
LIN {X -0.168,Y -658.932,Z 1359.400,A 0.000,B 0.000,C 90.000,E1 108.055} C_DIS
LIN {X 0.235,Y -662.977,Z 1359.395,A 0.000,B 0.000,C 90.000,E1 107.040} C_DIS
LIN {X 0.047,Y -664.825,Z 1359.392,A 0.000,B 0.000,C 90.000,E1 106.567} C_DIS
LIN {X -0.025,Y -667.296,Z 1359.388,A 0.000,B 0.000,C 90.000,E1 105.843} C_DIS
LIN {X -0.105,Y -668.076,Z 1359.387,A 0.000,B 0.000,C 90.000,E1 105.607} C_DIS
LIN {X -0.156,Y -669.841,Z 1359.383,A 0.000,B 0.000,C 90.000,E1 104.883} C_DIS
LIN {X 0.350,Y -670.811,Z 1359.380,A 0.000,B 0.000,C 90.000,E1 104.356} C_DIS
LIN {X 0.216,Y -671.537,Z 1359.377,A 0.000,B 0.000,C 90.000,E1 103.883} C_DIS
LIN {X 0.024,Y -672.244,Z 1359.373,A 0.000,B 0.000,C 90.000,E1 103.175} C_DIS
LIN {X -0.312,Y -672.465,Z 1359.369,A 0.000,B 0.000,C 90.000,E1 102.479} C_DIS
LIN {X 0.225,Y -672.439,Z 1359.367,A 0.000,B 0.000,C 90.000,E1 101.951} C_DIS
LIN {X 0.036,Y -671.929,Z 1359.363,A 0.000,B 0.000,C 90.000,E1 101.243} C_DIS
LIN {X -0.223,Y -671.396,Z 1359.360,A 0.000,B 0.000,C 90.000,E1 100.782} C_DIS
LIN {X 0.301,Y -670.659,Z 1359.357,A 0.000,B 0.000,C 90.000,E1 100.254} C_DIS
LIN {X 0.042,Y -669.660,Z 1359.354,A 0.000,B 0.000,C 90.000,E1 99.792} C_DIS
LIN {X -0.112,Y -668.392,Z 1359.352,A 0.000,B 0.000,C 90.000,E1 99.321} C_DIS
LIN {X 0.277,Y -666.833,Z 1359.349,A 0.000,B 0.000,C 90.000,E1 98.803} C_DIS
LIN {X -0.093,Y -664.099,Z 1359.345,A 0.000,B 0.000,C 90.000,E1 98.106} C_DIS
LIN {X 0.272,Y -662.087,Z 1359.342,A 0.000,B 0.000,C 90.000,E1 97.587} C_DIS
LIN {X -0.147,Y -658.635,Z 1359.338,A 0.000,B 0.000,C 90.000,E1 96.891} C_DIS
LIN {X -0.025,Y -654.923,Z 1359.334,A 0.000,B 0.000,C 90.000,E1 96.144} C_DIS
